(* LS Electric XG5000 project: HS(230517) *)
(* PLC NewPLC *)
(* module base 0 slot 0: FEnet:XGL-EFMT(B) (Fast Ethernet 통신 모듈, 전기 Master) *)
(* module base 1 slot 0: 아날로그입력 모듈:XGF-AC8A (A/D 전류 입력형 8채널) *)
(* module base 1 slot 1: 입력 모듈:XGI-D28A/B (DC 24V 입력, 64점 (전류소스 싱크공용/ 전류소스 입력)) *)
(* module base 1 slot 2: 입력 모듈:XGI-D28A/B (DC 24V 입력, 64점 (전류소스 싱크공용/ 전류소스 입력)) *)
(* module base 1 slot 3: 입력 모듈:XGI-D28A/B (DC 24V 입력, 64점 (전류소스 싱크공용/ 전류소스 입력)) *)
(* module base 1 slot 4: 출력 모듈:XGQ-TR8A/B (트랜지스터 출력, 64점 (0.1A용, 싱크출력/소스출력)) *)
(* module base 1 slot 5: 출력 모듈:XGQ-TR8A/B (트랜지스터 출력, 64점 (0.1A용, 싱크출력/소스출력)) *)
(* module base 1 slot 6: 출력 모듈:XGQ-TR8A/B (트랜지스터 출력, 64점 (0.1A용, 싱크출력/소스출력)) *)
VAR_GLOBAL
    _0100_CH0_ACT AT %UX1.0.16 : BOOL; (* 아날로그입력 모듈: 채널0 운전중 *)
    _0100_CH0_DATA AT %UW1.0.2 : INT; (* 아날로그입력 모듈: 채널0 변환값 *)
    _0100_CH0_IDD AT %UX1.0.160 : BOOL; (* 아날로그입력 모듈: 채널0 입력단선검출 *)
    _0100_CH1_ACT AT %UX1.0.17 : BOOL; (* 아날로그입력 모듈: 채널1 운전중 *)
    _0100_CH1_DATA AT %UW1.0.3 : INT; (* 아날로그입력 모듈: 채널1 변환값 *)
    _0100_CH1_IDD AT %UX1.0.161 : BOOL; (* 아날로그입력 모듈: 채널1 입력단선검출 *)
    _0100_CH2_ACT AT %UX1.0.18 : BOOL; (* 아날로그입력 모듈: 채널2 운전중 *)
    _0100_CH2_DATA AT %UW1.0.4 : INT; (* 아날로그입력 모듈: 채널2 변환값 *)
    _0100_CH2_IDD AT %UX1.0.162 : BOOL; (* 아날로그입력 모듈: 채널2 입력단선검출 *)
    _0100_CH3_ACT AT %UX1.0.19 : BOOL; (* 아날로그입력 모듈: 채널3 운전중 *)
    _0100_CH3_DATA AT %UW1.0.5 : INT; (* 아날로그입력 모듈: 채널3 변환값 *)
    _0100_CH3_IDD AT %UX1.0.163 : BOOL; (* 아날로그입력 모듈: 채널3 입력단선검출 *)
    _0100_CH4_ACT AT %UX1.0.20 : BOOL; (* 아날로그입력 모듈: 채널4 운전중 *)
    _0100_CH4_DATA AT %UW1.0.6 : INT; (* 아날로그입력 모듈: 채널4 변환값 *)
    _0100_CH4_IDD AT %UX1.0.164 : BOOL; (* 아날로그입력 모듈: 채널4 입력단선검출 *)
    _0100_CH5_ACT AT %UX1.0.21 : BOOL; (* 아날로그입력 모듈: 채널5 운전중 *)
    _0100_CH5_DATA AT %UW1.0.7 : INT; (* 아날로그입력 모듈: 채널5 변환값 *)
    _0100_CH5_IDD AT %UX1.0.165 : BOOL; (* 아날로그입력 모듈: 채널5 입력단선검출 *)
    _0100_CH6_ACT AT %UX1.0.22 : BOOL; (* 아날로그입력 모듈: 채널6 운전중 *)
    _0100_CH6_DATA AT %UW1.0.8 : INT; (* 아날로그입력 모듈: 채널6 변환값 *)
    _0100_CH6_IDD AT %UX1.0.166 : BOOL; (* 아날로그입력 모듈: 채널6 입력단선검출 *)
    _0100_CH7_ACT AT %UX1.0.23 : BOOL; (* 아날로그입력 모듈: 채널7 운전중 *)
    _0100_CH7_DATA AT %UW1.0.9 : INT; (* 아날로그입력 모듈: 채널7 변환값 *)
    _0100_CH7_IDD AT %UX1.0.167 : BOOL; (* 아날로그입력 모듈: 채널7 입력단선검출 *)
END_VAR

(* Comments on direct variables
%IX1.1.0	Power On_PB
%IX1.1.1	Power Off_PB
%IX1.1.2	TK1LK_On
%IX1.1.3	출하대 #2_EM
%IX1.1.4	FIRE_EM
SIG
%IX1.1.5	Manual_PB
%IX1.1.6	Auto_PB
%IX1.1.7	TRAIN EM
#1 SIG
%IX1.1.8	TRAIN EM
#2 SIG
%IX1.1.9	TRAIN EM
#3 SIG
%IX1.1.10	TRAIN EM
#4 SIG
%IX1.1.11	BCVF Trouble
%IX1.1.12	AUTO START PB
%IX1.1.13	AUTO Stop PB
%IX1.1.14	LAMP TEST PB
%IX1.1.15	EM-Reset [Panel]
%IX1.1.16	Buffer Tank_EM
%IX1.1.17	Main Tank_EM
%IX1.1.18	출하대 #1_EM
%IX1.1.19	Panel_EM
%IX1.1.20	Scada_선택
%IX1.1.21	Panel_선택
%IX1.1.22	Leakage-1 (L01301) On
%IX1.1.23	VENT1_On
%IX1.1.24	VENT1 Truble_On
%IX1.1.25	TK-001 Clearance
%IX1.1.26	P012A
 OCR & Thermostat
%IX1.1.27	P012A Local key Run[NC]
%IX1.1.28	P012A Stop_PB
%IX1.1.29	P012A Run_PB
%IX1.1.30	P012B
 OCR & Thermostat
%IX1.1.31	P012B Local ready[NC]
%IX1.1.32	P012B Stop_PB
%IX1.1.33	P012B Run_PB
%IX1.1.34	P013
 OCR & Thermostat
%IX1.1.35	P013 Local ready[NC]
%IX1.1.36	P013 Stop_PB
%IX1.1.37	P013 Run_PB
%IX1.1.38	P012A Flow s/w
%IX1.1.39	P012B Flow s/w
%IX1.1.40	P013 Flow Switch
%IX1.1.41	VENT2_On
%IX1.1.42	VENT2 Truble_On
%IX1.1.43	TK-002 Clearance
%IX1.1.44	P021A
 OCR & Thermostat
%IX1.1.45	P021A Local ready[NC]
%IX1.1.46	P021A Stop_PB
%IX1.1.47	P021A Run_PB
%IX1.1.48	P021B
 OCR & Thermostat
%IX1.1.49	P021B Local ready[NC]
%IX1.1.50	P021B Stop_PB
%IX1.1.51	P021B Run_PB
%IX1.1.52	P022
 OCR & Thermostat
%IX1.1.53	P022 Local SW
%IX1.1.54	P022 Stop_PB
%IX1.1.55	P022 Run_PB
%IX1.1.56	P021A Flow Switch
%IX1.1.57	P021B Flow Switch
%IX1.1.58	P022 Flow Switch
%IX1.1.59	TK002_HLV
%IX1.1.60	P012A 1차선택_PB
%IX1.1.61	P012A 2차선택_PB
%IX1.1.62	P012B 1차선택_PB
%IX1.1.63	P012B 2차선택_PB
%IX1.2.0	P021A 1차선택_PB
%IX1.2.1	P021A 2차선택_PB
%IX1.2.2	P021B 1차선택_PB
%IX1.2.3	P021B 2차선택_PB
%IX1.2.4	TK001_HLV
%IX1.2.5	TRANSFER
CLEARANCE
%IX1.2.6	P011A 
OCR & Thermostat
%IX1.2.7	P011A Local ready[NC]
%IX1.2.8	P011A Stop
[Panel]
%IX1.2.9	P011A Run
[Panel]
%IX1.2.10	P011B
 OCR & Thermostat
%IX1.2.11	P011B  Local ready[NC]
%IX1.2.12	P011B Stop_PB
%IX1.2.13	P011B Run_PB
%IX1.2.14	P011C
 OCR & Thermostat
%IX1.2.15	P011C Local ready[NC]
%IX1.2.16	P011C Stop_PB
%IX1.2.17	P011C Run_PB
%IX1.2.18	P011A Flow Switch
%IX1.2.19	P011B Flow Switch
%IX1.2.20	P011C Flow Switch
%IX1.2.21	P011A 1차 선택_PB
%IX1.2.22	P011A 2차선택_PB
%IX1.2.23	P011B 1차 선택_PB
%IX1.2.24	P011B 2차선택_PB
%IX1.2.25	P011C 1차선택_PB
%IX1.2.26	P011C 2차선택_PB
%IX1.2.27	Surge MOV_TR
%IX1.2.28	Surge MOV_LO
%IX1.2.29	Surge Close_PB
%IX1.2.30	Surge 
Close
Position
%IX1.2.31	Surge Open_PB
%IX1.2.32	Surge 
Open Position
%IX1.2.35	RTU-1 Close_PB
%IX1.2.37	RTU-1 Open_PB
%IX1.2.38	RTU-1 MOV_OP
%IX1.2.39	Transfer 수동_운전
%IX1.2.40	Transfer 자동_운전
%IX1.2.41	DR-Tank Water_On
%IX1.2.42	HLVD Close
%IX1.2.43	DRAIN
CLEARANCE
%IX1.2.44	P031
 OCR & Thermostat
%IX1.2.45	P031 Local SW
%IX1.2.46	P031 Stop_PB
%IX1.2.47	P031 Run_PB
%IX1.2.48	R2 PT201A-B 
%IX1.2.49	R3 FT201A-B
%IX1.2.50	R4 PT202A-B
%IX1.2.51	R5 FT202A-B
%IX1.2.52	CAM6_On
%IX1.2.53	드레인 P031_FS
%IX1.2.54	P031 Pressure  SW
%IX1.2.55	LDS ON 
SIG
%IX1.2.56	HLVB(하차 VALVE)
%IX1.2.57	PANTO 1 VPS
%IX1.2.58	PANTO 2 VPS
%IX1.2.59	LDS OFF SIG
%IX1.2.60	LDS EM(HS)
%IX1.2.61	Horn Rest PB
%IX1.3.0	P011A MC On SIG
%IX1.3.1	P011B MC On SIG
%IX1.3.2	P011C MC On SIG
%IX1.3.3	P012A MC On SIG
%IX1.3.4	P012B MC On SIG
%IX1.3.5	P013 MC On SIG
%IX1.3.6	P021A MC ON SIG
%IX1.3.7	P021B MC On SIG
%IX1.3.8	P022 MC On SIG
%IX1.3.9	DRAIN MC On SIG
%ID1.0.0	디지털_입력
%QX1.4.0	Power On_Lamp
%QX1.4.1	Power Off_Lamp
%QX1.4.2	Panel 선택 Lamp
%QX1.4.3	Scada 선택 Lamp
%QX1.4.4	TK3 누유 Lamp
%QX1.4.5	Manual_Lamp
%QX1.4.6	Auto_Lamp
%QX1.4.7	Auto Start Lamp
%QX1.4.8	Auto Stop Lamp
%QX1.4.9	Leakage TK-001 Lamp
%QX1.4.10	Leakage TK-002 Lamp
%QX1.4.11	Leakage TK-003 Lamp
%QX1.4.12	EM TK01 (BUFFER) Lamp
%QX1.4.13	EM TK02 (MAIN) Lamp
%QX1.4.14	Lamp Test Lamp
%QX1.4.15	PANTO 1  EM LAMP
%QX1.4.16	Horn Stop Lamp
%QX1.4.17	EM Panel Lamp
%QX1.4.18	PANTO 2 EM LAMP
%QX1.4.19	FIRE_EM
LAMP
%QX1.4.22	PIT201A Trouble Lamp
%QX1.4.23	PIT201B Trouble Lamp
%QX1.4.24	CVP OPEN LAMP
%QX1.4.25	EV OPEN LAMP
%QX1.4.26	PIT202A Trouble Lamp
%QX1.4.27	PIT202B Trouble Lamp
%QX1.4.28	FIT3 Trouble Lamp
%QX1.4.29	FIT4 Trouble Lamp
%QX1.4.30	Master_Plc Lamp
%QX1.4.31	Standby_  Plc Lamp
%QX1.4.32	EM-Stop Reset Lamp
%QX1.4.33	Leakage-1 Lamp
%QX1.4.34	VENT1 Trouble Lamp
%QX1.4.35	VENT1 Run Lamp
%QX1.4.36	P012A Trouble Lamp
%QX1.4.37	P012A Local Lamp
%QX1.4.38	P012A Stop Lamp
%QX1.4.39	P012A Run Lamp
%QX1.4.40	P012B Trouble Lamp
%QX1.4.41	P012B Local Lamp
%QX1.4.42	P012B Stop Lamp
%QX1.4.43	P012B Run Lamp
%QX1.4.44	P013 Trouble Lamp
%QX1.4.45	P013 Local Lamp
%QX1.4.46	P013 Stop Lamp
%QX1.4.47	P013 Run Lamp
%QX1.4.48	TK-001 Level_HH
%QX1.4.49	TK-001 Level_H
%QX1.4.50	TK-001 ATG TROUBLE
%QX1.4.51	TK-001 Level_L
%QX1.4.52	TK-001 Level_LL
%QX1.4.53	VENT2 Trouble Lamp
%QX1.4.54	VENT2 Run Lamp
%QX1.4.55	P021A Trouble Lamp
%QX1.4.56	P021A Local Lamp
%QX1.4.57	P021A Stop Lamp
%QX1.4.58	P021A Run Lamp
%QX1.4.59	P021B Trouble Lamp
%QX1.4.60	P021B Local Lamp
%QX1.4.61	P021B Stop Lamp
%QX1.4.62	P021B Run Lamp
%QX1.4.63	P022 Trouble Lamp
%QX1.5.0	P022 Local Lamp
%QX1.5.1	P022 Stop Lamp
%QX1.5.2	P022 Run Lamp
%QX1.5.3	TK-002 Level_HH
%QX1.5.4	TK-002 Level_H
%QX1.5.5	TK-002 ATG TROUBLE
%QX1.5.6	TK-002 Level_L
%QX1.5.7	TK-002 Level_LL
%QX1.5.8	HLV 01301 Lamp
%QX1.5.9	P012A 1차 선택 Lamp
%QX1.5.10	P012A 2차 선택 Lamp
%QX1.5.11	P012B 1차 선택 Lamp
%QX1.5.12	P012B 2차 선택 Lamp
%QX1.5.13	P021A 1차 선택 Lamp
%QX1.5.14	P021A 2차 선택 Lamp
%QX1.5.15	P021B 1차 선택 Lamp
%QX1.5.16	P021B 2차 선택 Lamp
%QX1.5.17	TK-001 HLV_Out
%QX1.5.18	P011A Trouble Lamp
%QX1.5.19	P011A Local Lamp
%QX1.5.20	P011A Stop Lamp
%QX1.5.21	P011A Run Lamp
%QX1.5.22	P011B Trouble Lamp
%QX1.5.23	P011B Local Lamp
%QX1.5.24	P011B Stop Lamp
%QX1.5.25	P011B Run Lamp
%QX1.5.26	P011C Trouble Lamp
%QX1.5.27	P011C Local Lamp
%QX1.5.28	P011C Stop Lamp
%QX1.5.29	P011C Run Lamp
%QX1.5.30	P011A 1차 선택 Lamp
%QX1.5.31	P011A 2차 선택 Lamp
%QX1.5.32	P011B 1차 선택 Lamp
%QX1.5.33	P011B 2차 선택 Lamp
%QX1.5.34	P011C 1차 선택 Lamp
%QX1.5.35	P011C 2차 선택 Lamp
%QX1.5.36	Surge Trouble Lamp
%QX1.5.38	Surge Close Lamp
%QX1.5.39	Surge 
Open Lamp
%QX1.5.40	RTU-1 Trouble Lamp
%QX1.5.41	RTU-1 Local Lamp
%QX1.5.42	RTU-1 Close Lamp
%QX1.5.43	RTU-1 Open Lamp
%QX1.5.44	Transfer 수동 LAMP
%QX1.5.45	Transfer 자동 LAMP
%QX1.5.46	600GPM LAMP
%QX1.5.47	1200GPM LAMP
%QX1.5.48	POLPRV LAMP
%QX1.5.49	RTU#1 OPEN LAMP
%QX1.5.50	RTU#2 OPEN LAMP
%QX1.5.51	RTU#3 OPEN LAMP
%QX1.5.52	RTU#4 OPEN LAMP
%QX1.5.53	RTU#5 OPEN LAMP
%QX1.5.54	Drain Water Lamp
%QX1.5.55	Drain HLVD_Full Lamp
%QX1.5.56	P031 Trouble Lamp
%QX1.5.57	P031 Local Lamp
%QX1.5.58	P031 Stop Lamp
%QX1.5.59	P031 Run Lamp
%QX1.5.60	TK-003 Level_HH
%QX1.5.61	TK-003 Level_H
%QX1.5.62	TK-003 ATG TROUBLE
%QX1.5.63	TK-003 Level_L
%QX1.6.0	TK-003 Level_LL
%QX1.6.1	CVP_Sol
%QX1.6.2	EV_Sol
%QX1.6.3	P011A_CVTF
%QX1.6.4	P011B_CVTF
%QX1.6.5	P011C_CVTF
%QX1.6.6	P-011A MCC_Run
%QX1.6.7	P-011B MCC_Run
%QX1.6.8	P-011C MCC_Run
%QX1.6.9	P-012A MCC_Run
%QX1.6.10	P-012B MCC_Run
%QX1.6.11	P-013 MCC_Run
%QX1.6.12	TK-001 HLV_Sol
%QX1.6.13	P-021A MCC_Run
%QX1.6.14	P-021B MCC_Run
%QX1.6.15	P-022 MCC_Run
%QX1.6.16	TK-001 HLV_Sol
%QX1.6.17	P-031 MCC_Run
%QX1.6.18	TK-003 HLVD_Out
%QX1.6.19	Surge Valve Open
%QX1.6.20	Surge Valve Close 
%QX1.6.21	RMOR
%QX1.6.22	RMCR
%QX1.6.23	Horn_Relay
%QX1.6.24	CVPl Lamp
%QX1.6.25	EV Lamp
%QX1.6.26	SURGE MOV
CLOSE SIG
%QX1.6.27	TRANSFER PUMP RUN
SIG
%QX1.6.28	SURGE MOV
OPEN SIG
%QX1.6.34	TO LDS
[SURGE CLOSE]
%QX1.6.35	TO LDS
[SURGE OPEN]
%QX1.6.36	TO LDS
[TP ALARM]
%QX1.6.37	LDS PUMP STOP SIG
%MX0	출하압력 Min
%MX1	TK01_EM
%MX2	TK02_EM
%MX3	PANTO 1 EM
%MX4	Panel_EM
%MX5	Total Em 
%MX6	Total Alarm
%MX7	Horn_Stop
%MX8	Horn Stop   Lamp   (SCADA)
%MX9	EM-Stop Reset   Lamp   (SCADA)
%MX10	P011A Pump Stop Set
%MX11	P011B Pump Stop Set
%MX12	P011C Pump Stop Set
%MX13	P012A Pump Stop Set
%MX14	P012B Pump Stop Set
%MX15	P013 Pump Stop Set
%MX16	LDS_EM(HS)
%MX17	LDS_EM
(POL)
%MX18	NMR5000_ERR
%MX19	FIRE_EM
%MX20	POL 수령탱크 HH
%MX21	P021A Pump Stop Set
%MX22	P021B Pump Stop Set
%MX23	P022 Pump Stop Set
%MX24	P031 Pump Stop Set
%MX25	P011A Lock key Run
%MX26	P011B Lock key Run
%MX27	P011C Lock key Run
%MX28	P012A Lock key Run
%MX29	P012B Lock key Run
%MX30	P013 Lock key Run
%MX31	P021A Lock key Run
%MX32	P021B Lock key Run
%MX33	P022 Lock key Run
%MX34	P031 Lock key Run
%MX41	POL TO RTU#1 ON SIG
%MX42	POL TO RTU#2 ON SIG
%MX43	POL TO RTU#3 ON SIG
%MX44	POL TO RTU#4 ON SIG
%MX45	POL TO RTU#5 ON SIG
%MX64	from SCADA  Manual [Select]
%MX65	from SCADA Auto [Select]
%MX66	AUTO START (SCADA)
%MX67	AUTO Stop PB(Scada)
%MX68	EM-Reset [SCADA]
%MX69	Horn Reset SCADA
%MX76	F03 Auto On_Out
%MX77	F03 Manual On_PB
%MX78	F03 Manual On_Out
%MX79	F01 Alam_Reset
%MX80	TRAIN EM
#1
%MX81	TRAIN EM
#2
%MX82	TRAIN EM
#3
%MX83	TRAIN EM
#4
%MX100	CH0 단선검출
%MX101	CH1 단선검출
%MX102	CH2 단선검출
%MX103	CH3 단선검출
%MX104	CH4 단선검출
%MX105	CH5 단선검출
%MX106	CH6 단선검출
%MX107	CH7 단선검출
%MX128	P011A Run [SCADA]
%MX129	P011A Stop
[SCADA]
%MX132	P011B Run [SCADA]
%MX133	P011B Stop_PB Scada
%MX136	P011C Run_PB Scada
%MX137	P011B Stop_PB Scada
%MX140	P012A Run_PB Scada
%MX141	P012A Stop_PB Scada
%MX144	P012B Run_PB Scada
%MX145	P012B Stop_PB Scada
%MX148	P013 Run_PB Scada
%MX149	P013 Stop_PB Scada
%MX152	P021A Run_PB Scada
%MX153	P021A Stop_PB Scada
%MX156	P021B Run_PB Scada
%MX157	P021B Stop_PB Scada
%MX160	P022 Run_PB Scada
%MX161	P022 Stop_PB Scada
%MX164	P031 Run_PB Scada
%MX165	P031 Stop_PB Scada
%MX266	MOV M01201 OPEN
%MX267	MOV M01201 CLOSE
%MX310	TK-001 Level_HH
%MX311	TK-001 Level_H
%MX312	TK-001 ATG TROUBLE SIG
%MX313	TK-001 Level_L
%MX314	TK-001 Level_LL
%MX320	TK-002 Level_HH
%MX321	TK-002 Level_H
%MX322	TK-002 ATG TROUBLE SIG
%MX323	TK-002 Level_L
%MX324	TK-002 Level_LL
%MX325	POL TOTAL EM (POL ->SCADA ->HS)
%MX330	TK-003 Level_HH
%MX331	TK-003 Level_H
%MX332	TK-003 ATG TROUBLE SIG
%MX333	TK-003 Level_L
%MX334	TK-003 Level_LL
%MX340	P011A 선택 SET
%MX341	P011B 선택 SET
%MX342	P011C 선택 SET
%MX343	P011A 2차 선택
%MX344	P011B 2차 선택
%MX345	P011C 2차 선택
%MX346	P011A 선택 SIG
%MX347	P011B 선택 SIG
%MX348	P011C 선택 SIG
%MX350	P012A 1차 선택
%MX351	P012B 1차 선택
%MX352	P012A 2차 선택
%MX353	P012B 2차 선택
%MX360	P021A 1차 선택
%MX361	P021B 1차 선택
%MX362	P021A 2차 선택
%MX363	P021B 2차 선택
%MX364	RTU1 OPEN LAMP (LDS->PLC)
%MX365	RTU2 OPEN LAMP (LDS->PLC)
%MX366	RTU3 OPEN LAMP (LDS->PLC)
%MX367	RTU4 OPEN LAMP (LDS->PLC)
%MX368	RTU5 OPEN LAMP (LDS->PLC)
%MX402	TK-110 ATG Trouble
%MX448	P011A  1차 선택 SWITCH  (SCADA)
%MX449	P011B 1차 선택 SWITCH  (SCADA)
%MX450	P011C 1차 선택 SWITCH  (SCADA)
%MX451	P011A  2차 선택 SWITCH  (SCADA)
%MX452	P011B 2차 선택 SWITCH  (SCADA)
%MX453	P011C 2차 선택 SWITCH  (SCADA)
%MX457	선택완료  (SCADA)
%MX458	P012A  1차 선택 SWITCH  (SCADA)
%MX459	P012B  1차 선택 SWITCH  (SCADA)
%MX460	P012A  2차 선택 SWITCH  (SCADA)
%MX461	P012B  2차 선택 SWITCH  (SCADA)
%MX467	선택완료  (SCADA)
%MX468	P021A  1차 선택 SWITCH  (SCADA)
%MX469	P021B 1차 선택 SWITCH  (SCADA)
%MX470	P021A  2차 선택 SWITCH  (SCADA)
%MX471	P021B 2차 선택 SWITCH  (SCADA)
%MX472	선택 완료    (SCADA)
%MX473	LDS 누유
%MX474	LDS  EM(POL)
%MX475	이송펌프 선택 초기화
%MX477	선택완료  (SCADA)
%MX960	P011A FS SIG
%MX961	P011B FS SIG
%MX962	P011C FS SIG
%MX963	P012A FS SIG
%MX964	P012B FS SIG
%MX965	P013 FS SIG
%MX966	P021A FS SIG
%MX967	P021B FS SIG
%MX968	P022 FS SIG
%MX969	P031 FS SIG
%MX1000	TK-002 MAIN TANK 누유
%MX1001	TK-001 BUFFER TANK 누유
%MX1002	TK-003 DRAIN TANK 누유
%MX6400	Panel Manual [Select]
%MX6401	SCADA  Manual [Select]
%MX6402	Panel   Auto [Select]
%MX6403	SCADA  Auto [Select]
%MX6410	Manual Select
[to SCADA]
%MX6411	Auto Select
[to SCADA]
%MX6464	LAMP TEST SIG
%MX6478	임시
%MX12800	PANTO 2 EM
%MX19200	P011A  Alarm
%MX19201	P011B  Alarm
%MX19202	P011C  Alarm
%MX19203	P012A  Alarm
%MX19204	P012B  Alarm
%MX19205	P013  Alarm
%MX19206	P021A  Alarm
%MX19207	P021B  Alarm
%MX19208	P022  Alarm
%MX19209	P031 Alarm
%MX19210	Surge Mov M01201 Trouble
%MX19211	RTU-1 Trouble Lamp(SCADA)
%MX19212	PIT201A Trouble   Lamp   (SCADA)
%MX19213	PIT201B Trouble   Lamp   (SCADA)
%MX19214	FIT201A Trouble   Lamp   (SCADA)
%MX19215	FIT201B Trouble   Lamp  (SCADA)
%MX19216	PIT202A Trouble   Lamp   (SCADA)
%MX19217	PIT202B Trouble   Lamp   (SCADA)
%MX19218	FIT3 Trouble   Lamp  (SCADA)
%MX19219	FIT4 Trouble   Lamp  (SCADA)
%MX19264	P011A RUN SIG
%MX19265	P011B 수동 RUN
%MX19266	P011C 수동 RUN
%MX19267	P012A 수동 RUN
%MX19268	P012B 수동 RUN
%MX19269	P013 수동 RUN
%MX19270	P021A 수동 RUN
%MX19271	P021B 수동 RUN
%MX19272	P022 수동 RUN
%MX19273	P031 수동 RUN
%MX19274	MOV 01201 OPEN 
%MX19275	MOV 01201 CLOSE
%MX19328	P011A FS ALARM
%MX19329	P011B FS ALARM
%MX19330	P011C FS ALARM
%MX19331	P012A FS ALARM
%MX19332	P012B FS ALARM
%MX19333	P013 FS ALARM
%MX19334	P021A FS ALARM
%MX19335	P021B FS ALARM
%MX19336	P022 FS ALARM
%MX19337	P031 FS ALARM
%MX23680	MAIN TANK 수령 송유관 색변화
%MX23681	MAIN TANK  불출 송유관 색변화
%MX23682	MAIN TANK  드레인 송유관 색변화 
%MX23683	BUFFER TANK  이송(BPCV) 송유관 색변화
%MX23684	BUFFER TANK이송  (CVTF1) 송유관 색변화
%MX23685	BUFFER TANK이송  (CVTF2) 송유관 색변화 2
%MX23686	BUFFER TANK이송  (CVTF3) 송유관 색변화
%MX23687	BUFFER TANK이송  (P012A,B) 송유관 색변화
%MX23688	BUFFER TANK회수 송유관 색변화1 
%MX23689	BUFFER TANK회수 송유관 색변화 2
%MX23691	BUFFER TANK DRAIN 송유관 색변화
%MX23692	BUFFER TANK 하차 송유관 색변화
%MX23693	DRAIN TANK DRAIN 송유관 색변화 5
%MX23694	PANTO1 송유관 색변화
%MX23695	PANTO02 송유관 색변화
%MX23696	이송 MAIN 송유관 색변화 
%MX23697	BUFFER & MAIN TANK DRAIN 송유관 색변화
%MX25600	AUTO START OK
%MX25601	AUTO START SIG
%MX25602	ALL REMOTE
%MX25603	AUTO START
%WB20	FROM POL
[HIGH 8 BIT]
%WB21	FROM POL
[LOW 8 BIT]
%WW0	TK-001 HH SET
%WW1	TK-001 H SET
%WW2	TK-001 L SET
%WW3	TK-001 LL SET
%WW4	TK-002 HH SET
%WW5	TK-002 H SET
%WW6	TK-002 L SET
%WW7	TK-002 LL SET
%WW9	FROM POL [16 BIT]
%WW10	이송 PUMP P011 1차 선택 SET
%WW11	이송 PUMP P011 2차 선택 SET
%WW12	이송 PUMP P012 1차 선택 SET
%WW13	이송 PUMP P012B  2차선택 SET
%WW14	이송 PUMP P021A  운전 선택 SET
%WW15	이송 PUMP P021B  운전 선택 SET
%WW20	TANK101 문자열
%WW21	TANK102 문자열
%WW22	TANK103 문자열
%WW30	TK-003 HH SET
%WW31	TK-003 H SET
%WW32	TK-003 L SET
%WW33	TK-003 LL SET
%WW34	P011 펌프 선택
%WW100	PT01 변환값
%WW102	PT01  이송압력 PSI
%WW150	P011A RUN SET
%WW151	P011B RUN SET
%WW152	P011C RUN SET
%WW153	P012A RUN SET
%WW154	P012B RUN SET
%WW155	P013 RUN SET
%WW156	P021A RUN SET
%WW157	P021B RUN SET
%WW158	P022 RUN SET
%WW159	P031 RUN SET
%WW160	MOV 01201 OPEN SET
%WW200	FT01 변환값
%WW202	FT01  이송유량 GPM
%WW300	PT02 변환값
%WW302	PT02  송유압력 PSI
%WW400	FT02 변환값
%WW402	FT02  이송유량 GPM
%WW500	DRAIN TANK 변환값
%WW506	DRAIN TANK LEVEL (PLC -> SCADA)
%WW600	MAIN TANK 변환값
%WW700	BUFFER TANK 변환값
%WW709	TK-110 ATG TROUBLE
%WW800	DRAIN TANK 변환값
%WW1000	TK-001 LEVEL 
(NMR TO PLC)
%WW1001	TK-001 ATG Trouble
%WW1003	TK-002 LEVEL (PLC->SCADA)
%WW1004	TK-002 ATG Trouble
*)

PROGRAM Main (* task: 스캔 프로그램 *)
VAR
    L_TST : TON;
    L_TST_FS : TON;
END_VAR

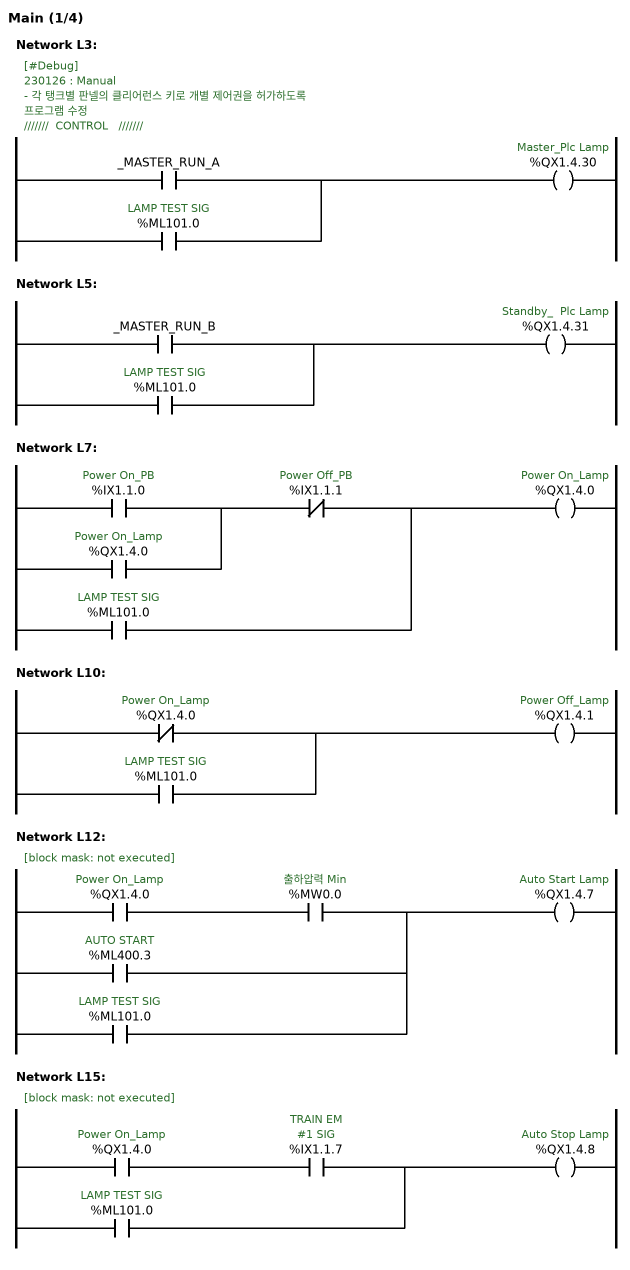
(* [#Debug] *)
(* 230126 : Manual / - 각 탱크별 판넬의 클리어런스 키로 개별 제어권을 허가하도록 / 프로그램 수정 *)
(* ///////  CONTROL   /////// *)
(* Rung L3 *)
%QX1.4.30 := _MASTER_RUN_A OR %ML101.0;
(* Rung L5 *)
%QX1.4.31 := _MASTER_RUN_B OR %ML101.0;
(* Rung L7 *)
%QX1.4.0 := ((%IX1.1.0 OR %QX1.4.0) AND NOT %IX1.1.1) OR %ML101.0;
(* Rung L10 *)
%QX1.4.1 := NOT %QX1.4.0 OR %ML101.0;
(* Rung L12 is block-masked: not executed *)
// %QX1.4.7 := (%QX1.4.0 AND %MW0.0) OR %ML400.3 OR %ML101.0;
(* Rung L15 is block-masked: not executed *)
// %QX1.4.8 := (%QX1.4.0 AND %IX1.1.7) OR %ML101.0;

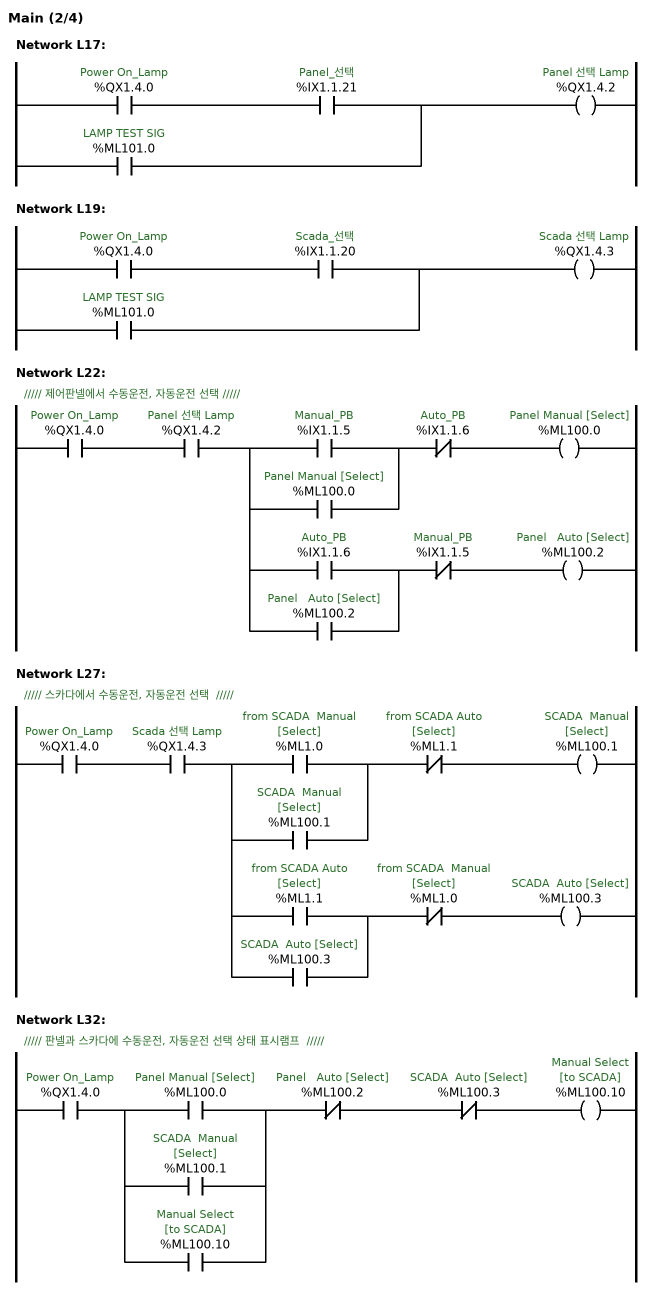
(* Rung L17 *)
%QX1.4.2 := (%QX1.4.0 AND %IX1.1.21) OR %ML101.0;
(* Rung L19 *)
%QX1.4.3 := (%QX1.4.0 AND %IX1.1.20) OR %ML101.0;
(* ///// 제어판넬에서 수동운전, 자동운전 선택 ///// *)
(* Rung L22 *)
%ML100.0 := %QX1.4.0 AND %QX1.4.2 AND (%IX1.1.5 OR %ML100.0) AND NOT %IX1.1.6;
%ML100.2 := %QX1.4.0 AND %QX1.4.2 AND (%IX1.1.6 OR %ML100.2) AND NOT %IX1.1.5;
(* ///// 스카다에서 수동운전, 자동운전 선택  ///// *)
(* Rung L27 *)
%ML100.1 := %QX1.4.0 AND %QX1.4.3 AND (%ML1.0 OR %ML100.1) AND NOT %ML1.1;
%ML100.3 := %QX1.4.0 AND %QX1.4.3 AND (%ML1.1 OR %ML100.3) AND NOT %ML1.0;
(* ///// 판넬과 스카다에 수동운전, 자동운전 선택 상태 표시램프  ///// *)
(* Rung L32 *)
%ML100.10 := %QX1.4.0 AND (%ML100.0 OR %ML100.1 OR %ML100.10) AND NOT %ML100.2 AND NOT %ML100.3;

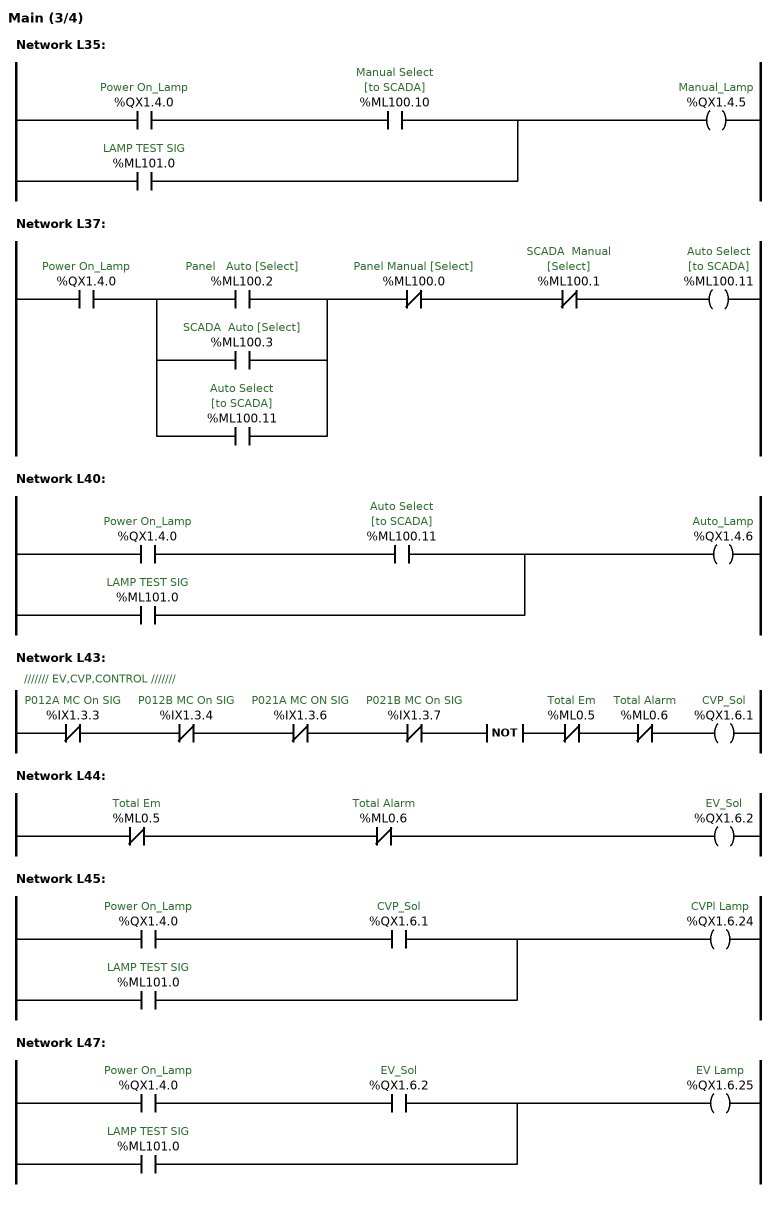
(* Rung L35 *)
%QX1.4.5 := (%QX1.4.0 AND %ML100.10) OR %ML101.0;
(* Rung L37 *)
%ML100.11 := %QX1.4.0 AND (%ML100.2 OR %ML100.3 OR %ML100.11) AND NOT %ML100.0 AND NOT %ML100.1;
(* Rung L40 *)
%QX1.4.6 := (%QX1.4.0 AND %ML100.11) OR %ML101.0;
(* /////// EV,CVP,CONTROL /////// *)
(* Rung L43 *)
%QX1.6.1 := NOT (NOT %IX1.3.3 AND NOT %IX1.3.4 AND NOT %IX1.3.6 AND NOT %IX1.3.7) AND NOT %ML0.5 AND NOT %ML0.6;
(* Rung L44 *)
%QX1.6.2 := NOT %ML0.5 AND NOT %ML0.6;
(* Rung L45 *)
%QX1.6.24 := (%QX1.4.0 AND %QX1.6.1) OR %ML101.0;
(* Rung L47 *)
%QX1.6.25 := (%QX1.4.0 AND %QX1.6.2) OR %ML101.0;

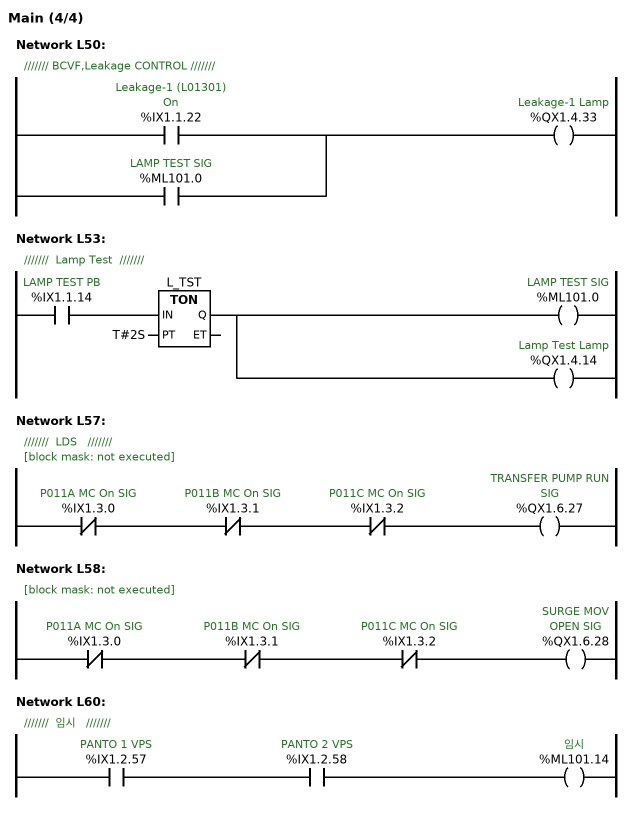
(* /////// BCVF,Leakage CONTROL /////// *)
(* Rung L50 *)
%QX1.4.33 := %IX1.1.22 OR %ML101.0;
(* ///////  Lamp Test  /////// *)
(* Rung L53 *)
L_TST(IN := %IX1.1.14, PT := T#2S);
%ML101.0 := L_TST.Q;
%QX1.4.14 := L_TST.Q;
(* ///////  LDS   /////// *)
(* Rung L57 is block-masked: not executed *)
// %QX1.6.27 := NOT %IX1.3.0 AND NOT %IX1.3.1 AND NOT %IX1.3.2;
(* Rung L58 is block-masked: not executed *)
// %QX1.6.28 := NOT %IX1.3.0 AND NOT %IX1.3.1 AND NOT %IX1.3.2;
(* ///////  임시   /////// *)
(* Rung L60 *)
%ML101.14 := %IX1.2.57 AND %IX1.2.58;
END_PROGRAM

PROGRAM Manual (* task: 스캔 프로그램 *)
VAR
    INST : TP; (* PUMP FS 떨림방지 *)
    INST1 : TP; (* PUMP FS 떨림방지 *)
    P011A_FS : TON;
    P011B_FS : TON;
    P011C_FS : TON;
    P012A_FS : TON;
    P012B_FS : TON;
    P012C_FS : TON;
    P013B_FS : TON;
    P013C_FS : TON;
    P013_FS : TON;
    P014_FS : TON;
    P021A_FS : TON;
    P022A_FS : TON;
    P022_FS : TON;
    P023_FS : TON;
    P031_FS : TON;
    P031_run : TON;
    P031_압력SW : TON;
    P032_FS : TON;
    P033_FS : TON;
    P034_FS : TON;
    P1O1B_FS : TON;
    P1O2B_FS : TON;
    P1O3B_FS : TON;
    TK031_HLV_Pressure_Charging : TON; (* 드레인탱크 031 HLVD 작동을 위한 상시 가압 탱크에 압력을 자체 충전하기위한 압력 감지 접점이 작동하면 펌프를 0.5초 지연 후 작동시킨다 *)
END_VAR
VAR_EXTERNAL
    _0100_CH2_DATA : INT; (* AT %UW1.0.4 *) (* 아날로그입력 모듈: 채널2 변환값 *)
    _0100_CH3_DATA : INT; (* AT %UW1.0.5 *) (* 아날로그입력 모듈: 채널3 변환값 *)
    _0100_CH4_ACT : BOOL; (* AT %UX1.0.20 *) (* 아날로그입력 모듈: 채널4 운전중 *)
    _0100_CH4_DATA : INT; (* AT %UW1.0.6 *) (* 아날로그입력 모듈: 채널4 변환값 *)
    _0100_CH5_ACT : BOOL; (* AT %UX1.0.21 *) (* 아날로그입력 모듈: 채널5 운전중 *)
    _0100_CH5_DATA : INT; (* AT %UW1.0.7 *) (* 아날로그입력 모듈: 채널5 변환값 *)
    _0100_CH6_ACT : BOOL; (* AT %UX1.0.22 *) (* 아날로그입력 모듈: 채널6 운전중 *)
    _0100_CH6_DATA : INT; (* AT %UW1.0.8 *) (* 아날로그입력 모듈: 채널6 변환값 *)
    _0100_CH7_ACT : BOOL; (* AT %UX1.0.23 *) (* 아날로그입력 모듈: 채널7 운전중 *)
    _0100_CH7_DATA : INT; (* AT %UW1.0.9 *) (* 아날로그입력 모듈: 채널7 변환값 *)
END_VAR
VAR
    _e1 : R_TRIG;
    _e2 : R_TRIG;
END_VAR

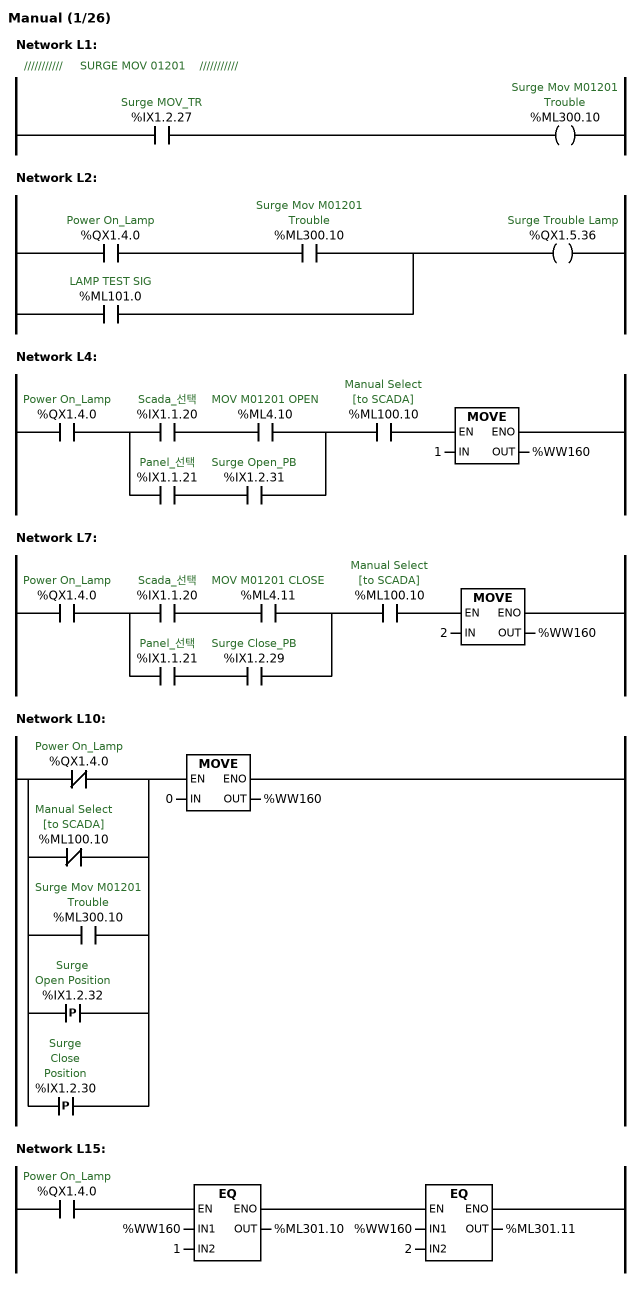
(* ///////////     SURGE MOV 01201    /////////// *)
(* Rung L1 *)
%ML300.10 := %IX1.2.27;
(* Rung L2 *)
%QX1.5.36 := (%QX1.4.0 AND %ML300.10) OR %ML101.0;
(* Rung L4 *)
IF %QX1.4.0 AND ((%IX1.1.20 AND %ML4.10) OR (%IX1.1.21 AND %IX1.2.31)) AND %ML100.10 THEN
    %WW160 := 1;
END_IF;
(* Rung L7 *)
IF %QX1.4.0 AND ((%IX1.1.20 AND %ML4.11) OR (%IX1.1.21 AND %IX1.2.29)) AND %ML100.10 THEN
    %WW160 := 2;
END_IF;
(* Rung L10 *)
_e1(CLK := %IX1.2.32);
_e2(CLK := %IX1.2.30);
IF NOT %QX1.4.0 OR NOT %ML100.10 OR %ML300.10 OR _e1.Q OR _e2.Q THEN %WW160 := 0; END_IF;
(* Rung L15 *)
IF %QX1.4.0 THEN
    %ML301.10 := %WW160 = 1;
    %ML301.11 := %WW160 = 2;
END_IF;

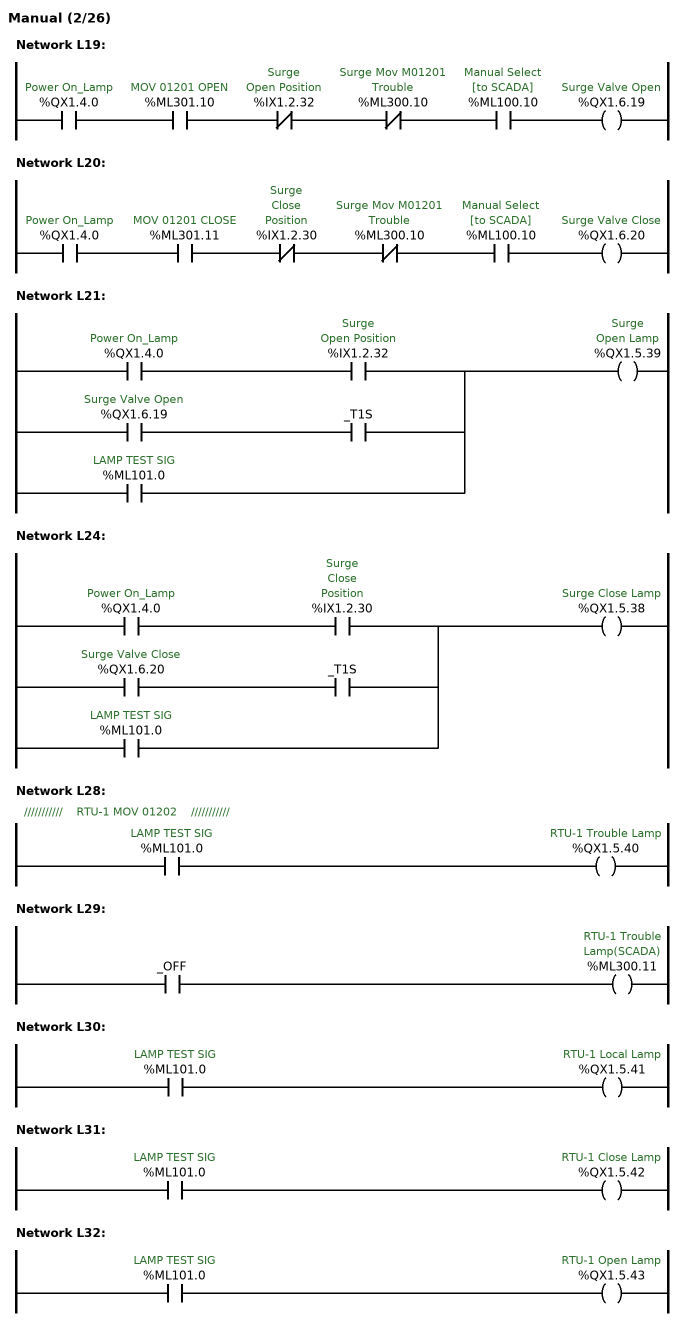
(* Rung L19 *)
%QX1.6.19 := %QX1.4.0 AND %ML301.10 AND NOT %IX1.2.32 AND NOT %ML300.10 AND %ML100.10;
(* Rung L20 *)
%QX1.6.20 := %QX1.4.0 AND %ML301.11 AND NOT %IX1.2.30 AND NOT %ML300.10 AND %ML100.10;
(* Rung L21 *)
%QX1.5.39 := (%QX1.4.0 AND %IX1.2.32) OR (%QX1.6.19 AND _T1S) OR %ML101.0;
(* Rung L24 *)
%QX1.5.38 := (%QX1.4.0 AND %IX1.2.30) OR (%QX1.6.20 AND _T1S) OR %ML101.0;
(* ///////////    RTU-1 MOV 01202    /////////// *)
(* Rung L28 *)
%QX1.5.40 := %ML101.0;
(* Rung L29 *)
%ML300.11 := _OFF;
(* Rung L30 *)
%QX1.5.41 := %ML101.0;
(* Rung L31 *)
%QX1.5.42 := %ML101.0;
(* Rung L32 *)
%QX1.5.43 := %ML101.0;

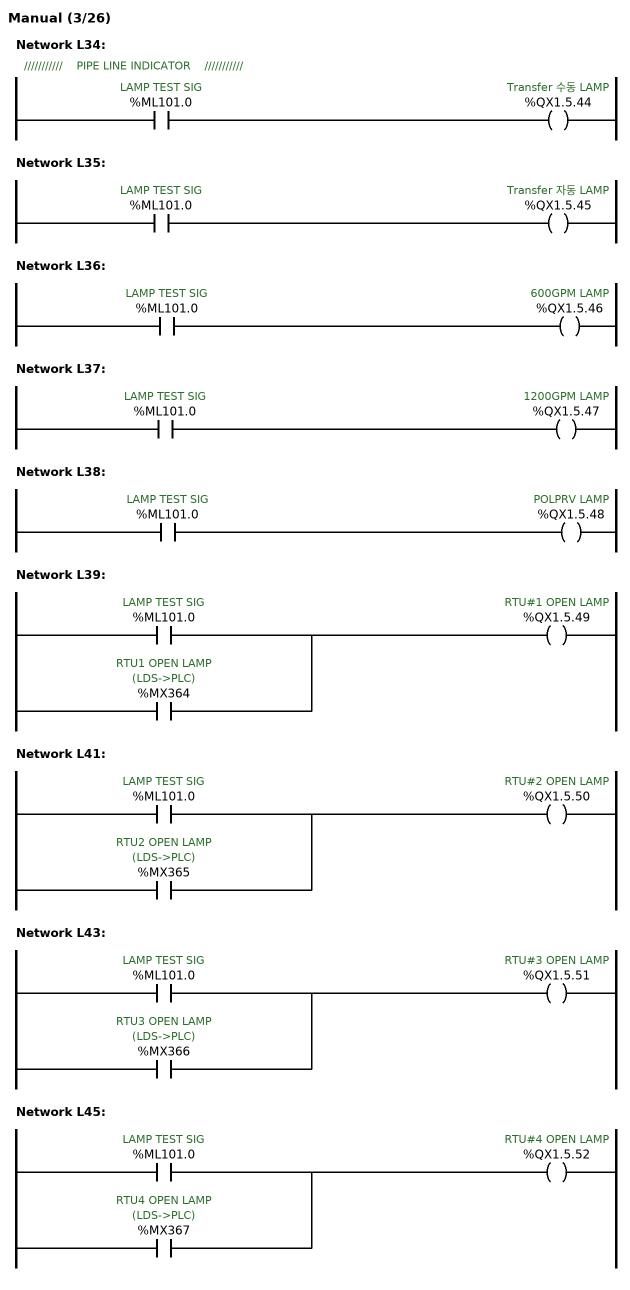
(* ///////////    PIPE LINE INDICATOR    /////////// *)
(* Rung L34 *)
%QX1.5.44 := %ML101.0;
(* Rung L35 *)
%QX1.5.45 := %ML101.0;
(* Rung L36 *)
%QX1.5.46 := %ML101.0;
(* Rung L37 *)
%QX1.5.47 := %ML101.0;
(* Rung L38 *)
%QX1.5.48 := %ML101.0;
(* Rung L39 *)
%QX1.5.49 := %ML101.0 OR %MX364;
(* Rung L41 *)
%QX1.5.50 := %ML101.0 OR %MX365;
(* Rung L43 *)
%QX1.5.51 := %ML101.0 OR %MX366;
(* Rung L45 *)
%QX1.5.52 := %ML101.0 OR %MX367;

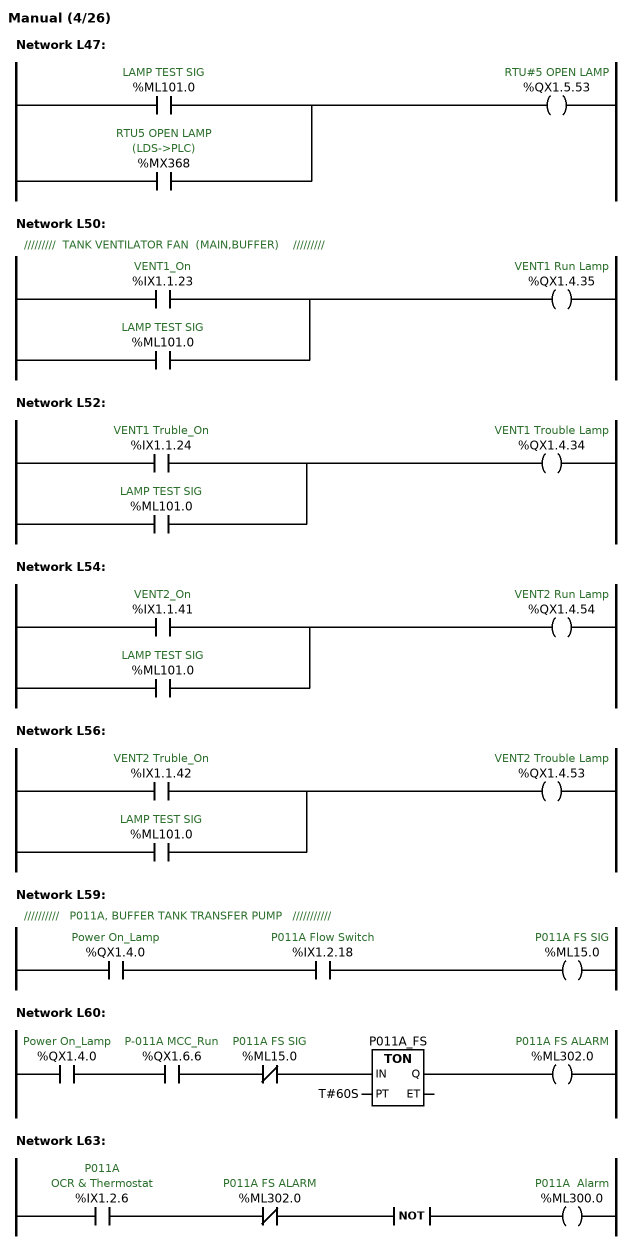
(* Rung L47 *)
%QX1.5.53 := %ML101.0 OR %MX368;
(* /////////  TANK VENTILATOR FAN  (MAIN,BUFFER)    ///////// *)
(* Rung L50 *)
%QX1.4.35 := %IX1.1.23 OR %ML101.0;
(* Rung L52 *)
%QX1.4.34 := %IX1.1.24 OR %ML101.0;
(* Rung L54 *)
%QX1.4.54 := %IX1.1.41 OR %ML101.0;
(* Rung L56 *)
%QX1.4.53 := %IX1.1.42 OR %ML101.0;
(* //////////   P011A, BUFFER TANK TRANSFER PUMP   /////////// *)
(* Rung L59 *)
%ML15.0 := %QX1.4.0 AND %IX1.2.18;
(* Rung L60 *)
P011A_FS(IN := %QX1.4.0 AND %QX1.6.6 AND NOT %ML15.0, PT := T#60S);
%ML302.0 := P011A_FS.Q;
(* Rung L63 *)
%ML300.0 := NOT (%IX1.2.6 AND NOT %ML302.0);

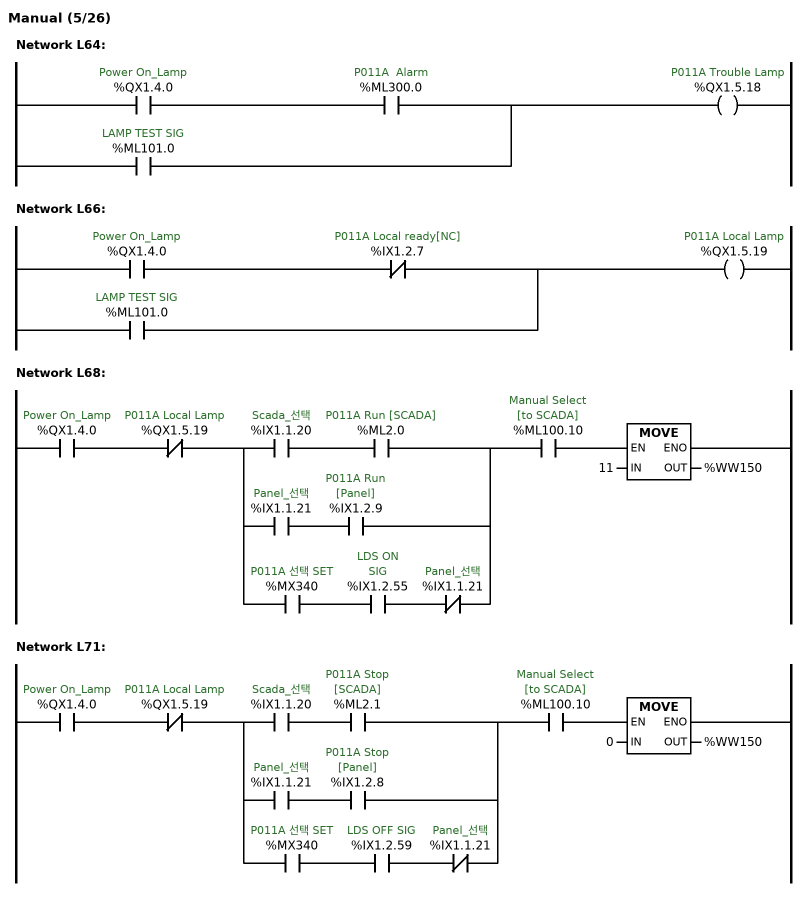
(* Rung L64 *)
%QX1.5.18 := (%QX1.4.0 AND %ML300.0) OR %ML101.0;
(* Rung L66 *)
%QX1.5.19 := (%QX1.4.0 AND NOT %IX1.2.7) OR %ML101.0;
(* Rung L68 *)
IF %QX1.4.0 AND NOT %QX1.5.19 AND ((%IX1.1.20 AND %ML2.0) OR (%IX1.1.21 AND %IX1.2.9) OR (%MX340 AND %IX1.2.55 AND NOT %IX1.1.21)) AND %ML100.10 THEN
    %WW150 := 11;
END_IF;
(* Rung L71 *)
IF %QX1.4.0 AND NOT %QX1.5.19 AND ((%IX1.1.20 AND %ML2.1) OR (%IX1.1.21 AND %IX1.2.8) OR (%MX340 AND %IX1.2.59 AND NOT %IX1.1.21)) AND %ML100.10 THEN
    %WW150 := 0;
END_IF;

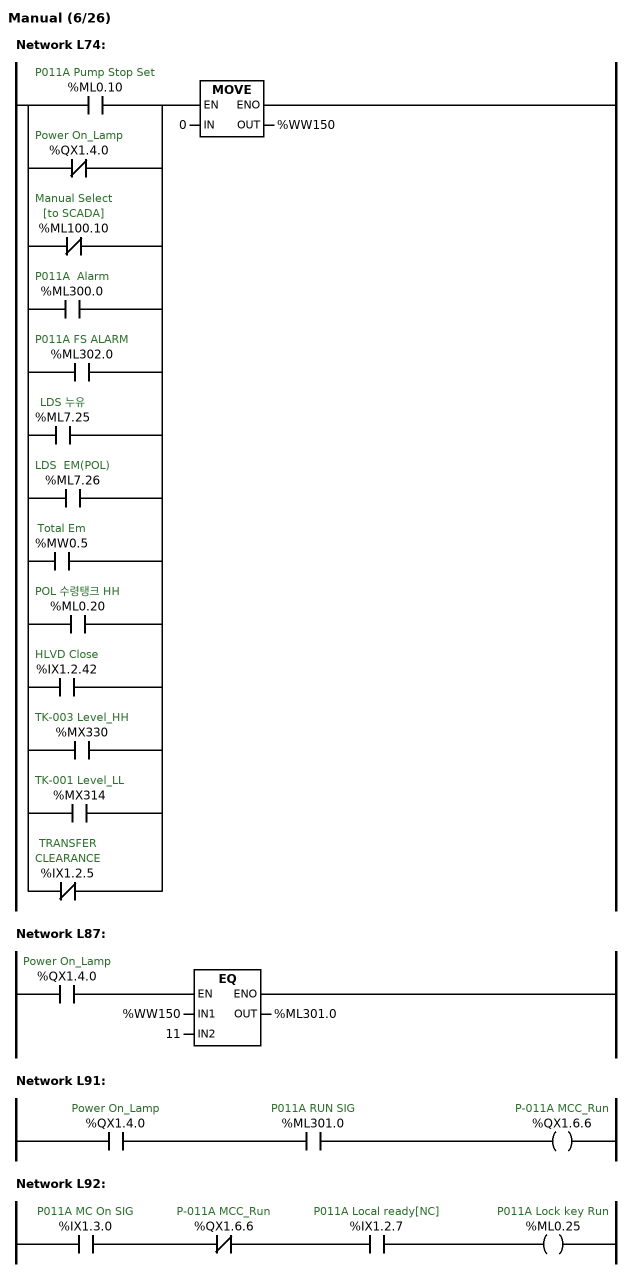
(* Rung L74 *)
IF %ML0.10 OR NOT %QX1.4.0 OR NOT %ML100.10 OR %ML300.0 OR %ML302.0 OR %ML7.25 OR %ML7.26 OR %MW0.5 OR %ML0.20 OR %IX1.2.42 OR %MX330 OR %MX314 OR NOT %IX1.2.5 THEN
    %WW150 := 0;
END_IF;
(* Rung L87 *)
IF %QX1.4.0 THEN %ML301.0 := %WW150 = 11; END_IF;
(* Rung L91 *)
%QX1.6.6 := %QX1.4.0 AND %ML301.0;
(* Rung L92 *)
%ML0.25 := %IX1.3.0 AND NOT %QX1.6.6 AND %IX1.2.7;

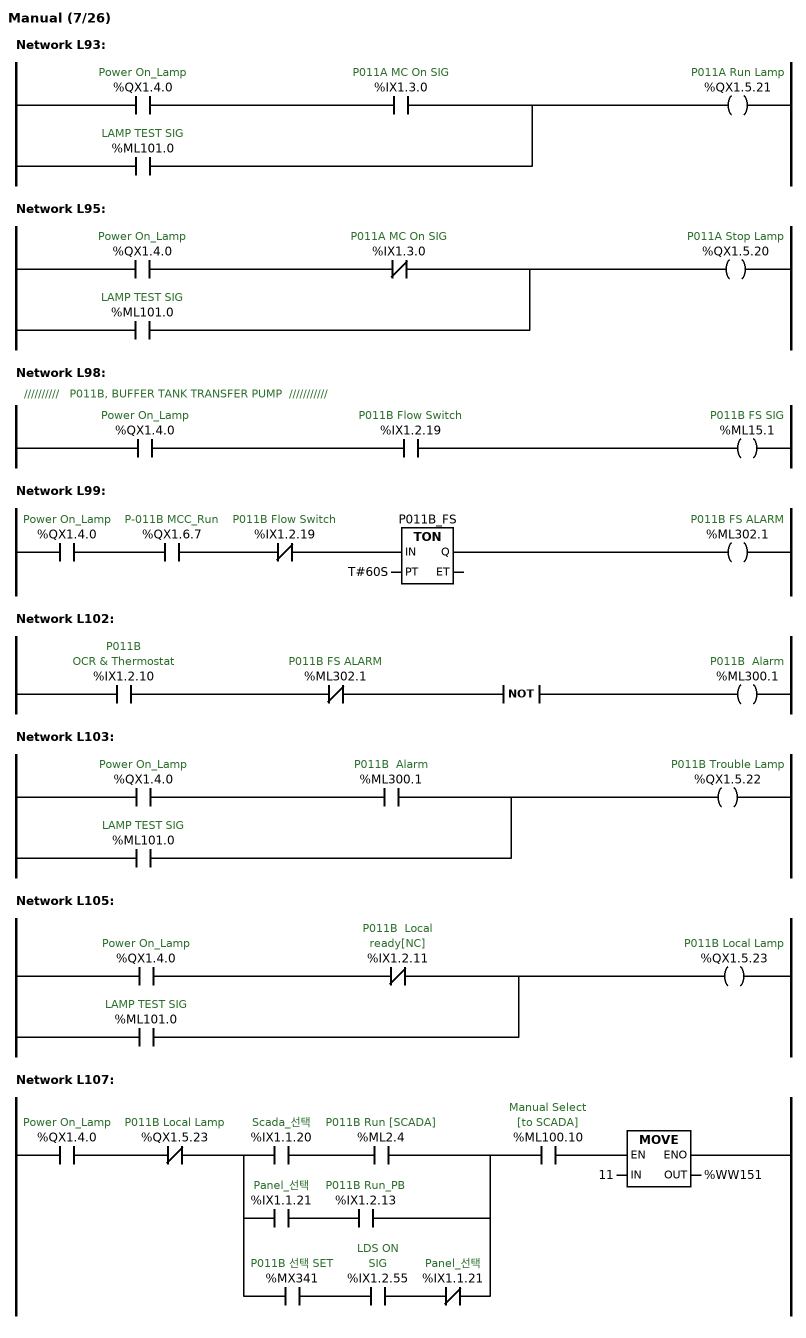
(* Rung L93 *)
%QX1.5.21 := (%QX1.4.0 AND %IX1.3.0) OR %ML101.0;
(* Rung L95 *)
%QX1.5.20 := (%QX1.4.0 AND NOT %IX1.3.0) OR %ML101.0;
(* //////////   P011B, BUFFER TANK TRANSFER PUMP  /////////// *)
(* Rung L98 *)
%ML15.1 := %QX1.4.0 AND %IX1.2.19;
(* Rung L99 *)
P011B_FS(IN := %QX1.4.0 AND %QX1.6.7 AND NOT %IX1.2.19, PT := T#60S);
%ML302.1 := P011B_FS.Q;
(* Rung L102 *)
%ML300.1 := NOT (%IX1.2.10 AND NOT %ML302.1);
(* Rung L103 *)
%QX1.5.22 := (%QX1.4.0 AND %ML300.1) OR %ML101.0;
(* Rung L105 *)
%QX1.5.23 := (%QX1.4.0 AND NOT %IX1.2.11) OR %ML101.0;
(* Rung L107 *)
IF %QX1.4.0 AND NOT %QX1.5.23 AND ((%IX1.1.20 AND %ML2.4) OR (%IX1.1.21 AND %IX1.2.13) OR (%MX341 AND %IX1.2.55 AND NOT %IX1.1.21)) AND %ML100.10 THEN
    %WW151 := 11;
END_IF;

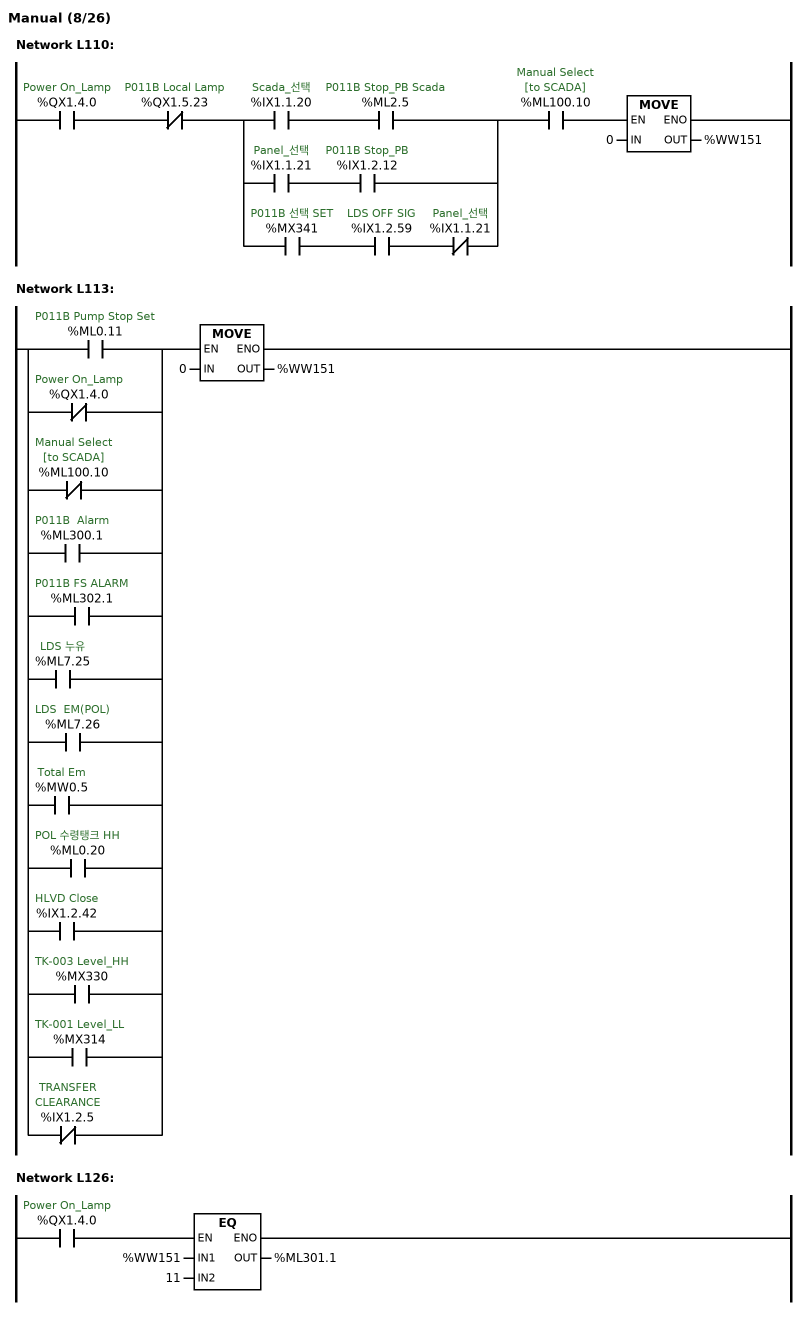
(* Rung L110 *)
IF %QX1.4.0 AND NOT %QX1.5.23 AND ((%IX1.1.20 AND %ML2.5) OR (%IX1.1.21 AND %IX1.2.12) OR (%MX341 AND %IX1.2.59 AND NOT %IX1.1.21)) AND %ML100.10 THEN
    %WW151 := 0;
END_IF;
(* Rung L113 *)
IF %ML0.11 OR NOT %QX1.4.0 OR NOT %ML100.10 OR %ML300.1 OR %ML302.1 OR %ML7.25 OR %ML7.26 OR %MW0.5 OR %ML0.20 OR %IX1.2.42 OR %MX330 OR %MX314 OR NOT %IX1.2.5 THEN
    %WW151 := 0;
END_IF;
(* Rung L126 *)
IF %QX1.4.0 THEN %ML301.1 := %WW151 = 11; END_IF;

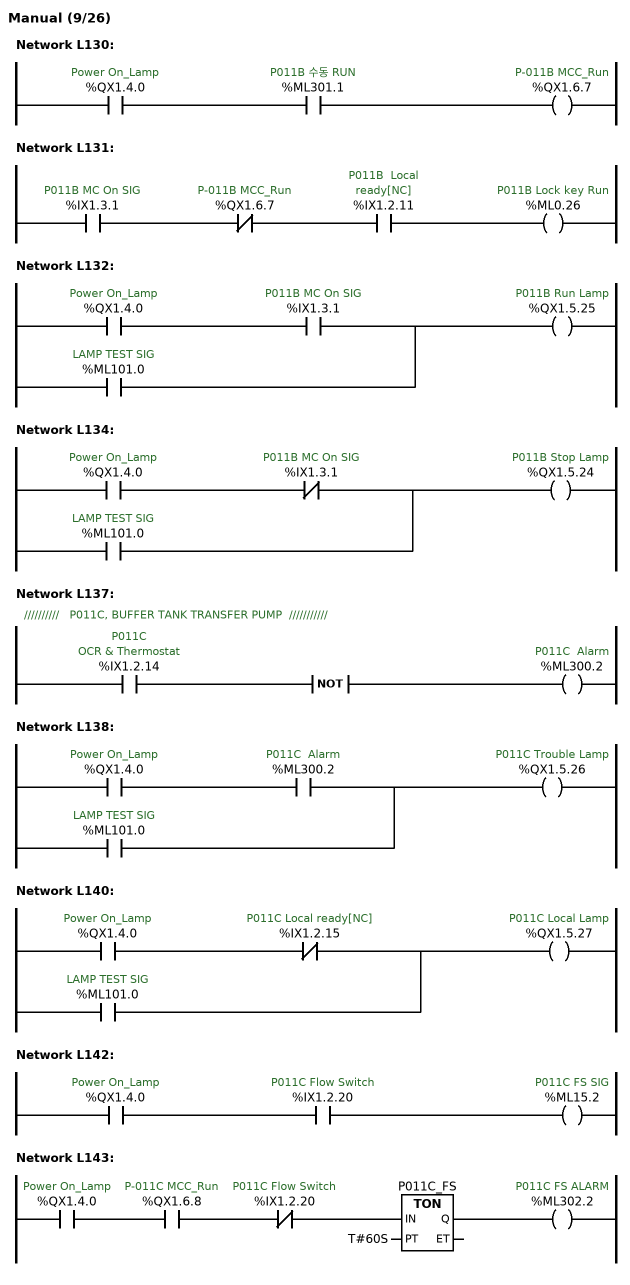
(* Rung L130 *)
%QX1.6.7 := %QX1.4.0 AND %ML301.1;
(* Rung L131 *)
%ML0.26 := %IX1.3.1 AND NOT %QX1.6.7 AND %IX1.2.11;
(* Rung L132 *)
%QX1.5.25 := (%QX1.4.0 AND %IX1.3.1) OR %ML101.0;
(* Rung L134 *)
%QX1.5.24 := (%QX1.4.0 AND NOT %IX1.3.1) OR %ML101.0;
(* //////////   P011C, BUFFER TANK TRANSFER PUMP  /////////// *)
(* Rung L137 *)
%ML300.2 := NOT %IX1.2.14;
(* Rung L138 *)
%QX1.5.26 := (%QX1.4.0 AND %ML300.2) OR %ML101.0;
(* Rung L140 *)
%QX1.5.27 := (%QX1.4.0 AND NOT %IX1.2.15) OR %ML101.0;
(* Rung L142 *)
%ML15.2 := %QX1.4.0 AND %IX1.2.20;
(* Rung L143 *)
P011C_FS(IN := %QX1.4.0 AND %QX1.6.8 AND NOT %IX1.2.20, PT := T#60S);
%ML302.2 := P011C_FS.Q;

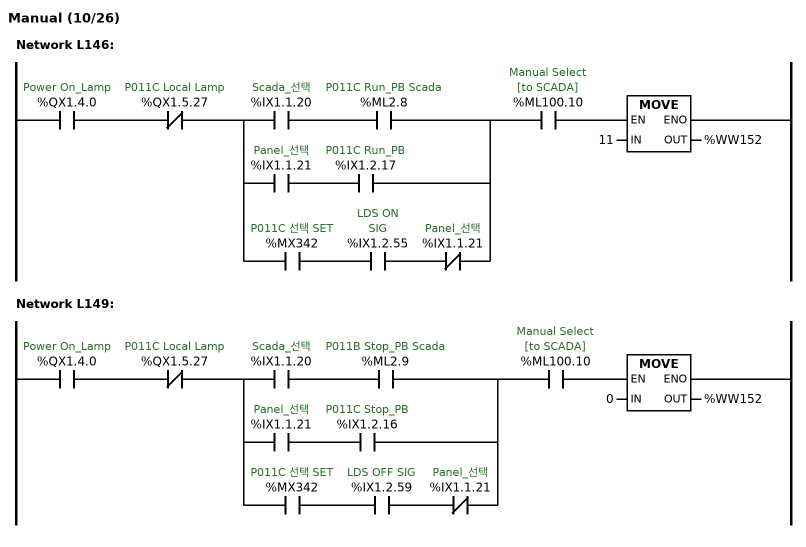
(* Rung L146 *)
IF %QX1.4.0 AND NOT %QX1.5.27 AND ((%IX1.1.20 AND %ML2.8) OR (%IX1.1.21 AND %IX1.2.17) OR (%MX342 AND %IX1.2.55 AND NOT %IX1.1.21)) AND %ML100.10 THEN
    %WW152 := 11;
END_IF;
(* Rung L149 *)
IF %QX1.4.0 AND NOT %QX1.5.27 AND ((%IX1.1.20 AND %ML2.9) OR (%IX1.1.21 AND %IX1.2.16) OR (%MX342 AND %IX1.2.59 AND NOT %IX1.1.21)) AND %ML100.10 THEN
    %WW152 := 0;
END_IF;

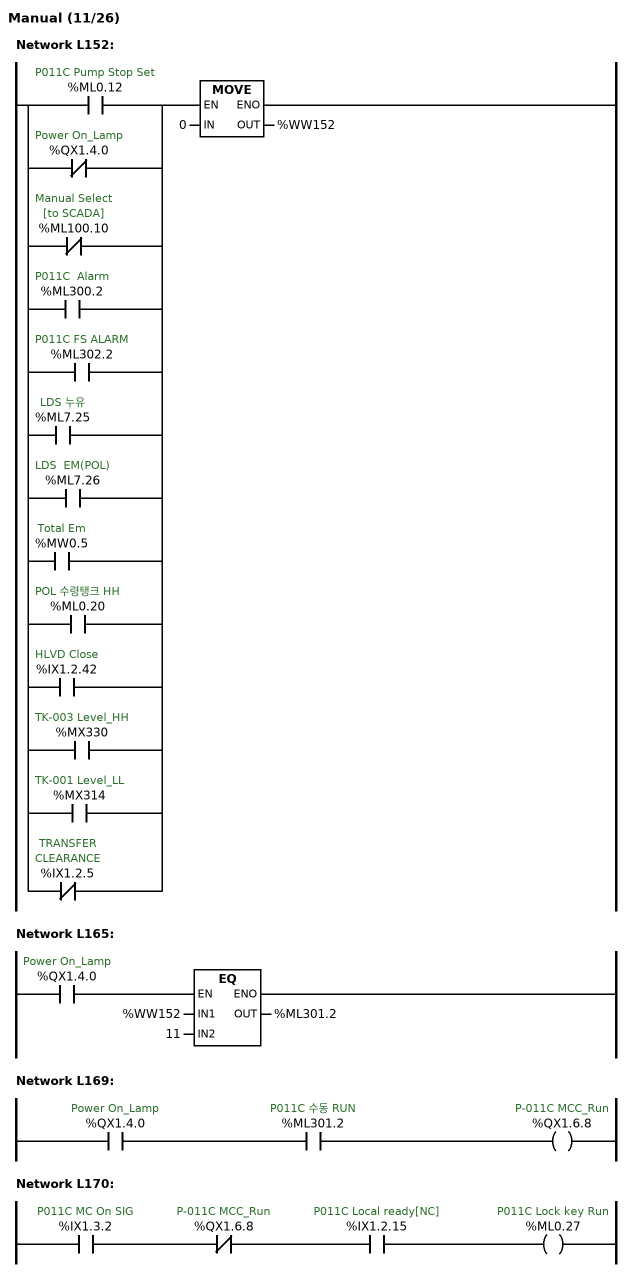
(* Rung L152 *)
IF %ML0.12 OR NOT %QX1.4.0 OR NOT %ML100.10 OR %ML300.2 OR %ML302.2 OR %ML7.25 OR %ML7.26 OR %MW0.5 OR %ML0.20 OR %IX1.2.42 OR %MX330 OR %MX314 OR NOT %IX1.2.5 THEN
    %WW152 := 0;
END_IF;
(* Rung L165 *)
IF %QX1.4.0 THEN %ML301.2 := %WW152 = 11; END_IF;
(* Rung L169 *)
%QX1.6.8 := %QX1.4.0 AND %ML301.2;
(* Rung L170 *)
%ML0.27 := %IX1.3.2 AND NOT %QX1.6.8 AND %IX1.2.15;

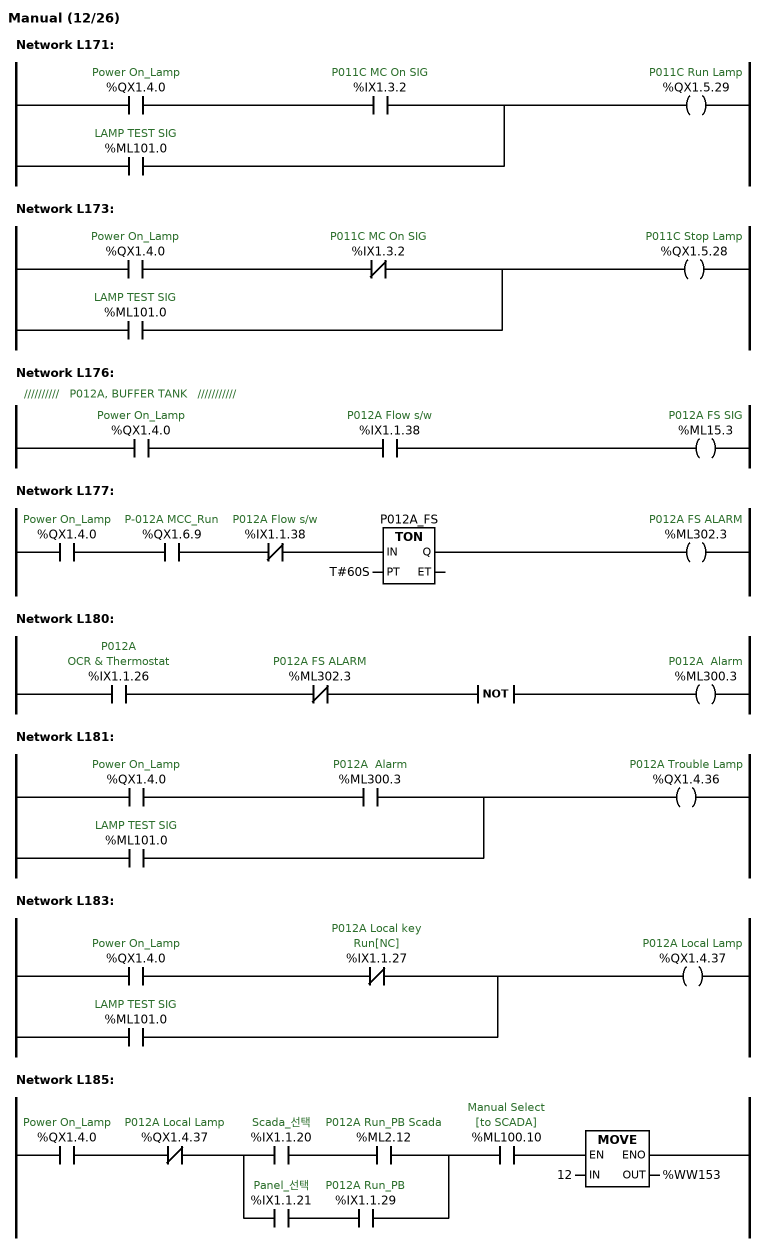
(* Rung L171 *)
%QX1.5.29 := (%QX1.4.0 AND %IX1.3.2) OR %ML101.0;
(* Rung L173 *)
%QX1.5.28 := (%QX1.4.0 AND NOT %IX1.3.2) OR %ML101.0;
(* //////////   P012A, BUFFER TANK   /////////// *)
(* Rung L176 *)
%ML15.3 := %QX1.4.0 AND %IX1.1.38;
(* Rung L177 *)
P012A_FS(IN := %QX1.4.0 AND %QX1.6.9 AND NOT %IX1.1.38, PT := T#60S);
%ML302.3 := P012A_FS.Q;
(* Rung L180 *)
%ML300.3 := NOT (%IX1.1.26 AND NOT %ML302.3);
(* Rung L181 *)
%QX1.4.36 := (%QX1.4.0 AND %ML300.3) OR %ML101.0;
(* Rung L183 *)
%QX1.4.37 := (%QX1.4.0 AND NOT %IX1.1.27) OR %ML101.0;
(* Rung L185 *)
IF %QX1.4.0 AND NOT %QX1.4.37 AND ((%IX1.1.20 AND %ML2.12) OR (%IX1.1.21 AND %IX1.1.29)) AND %ML100.10 THEN
    %WW153 := 12;
END_IF;

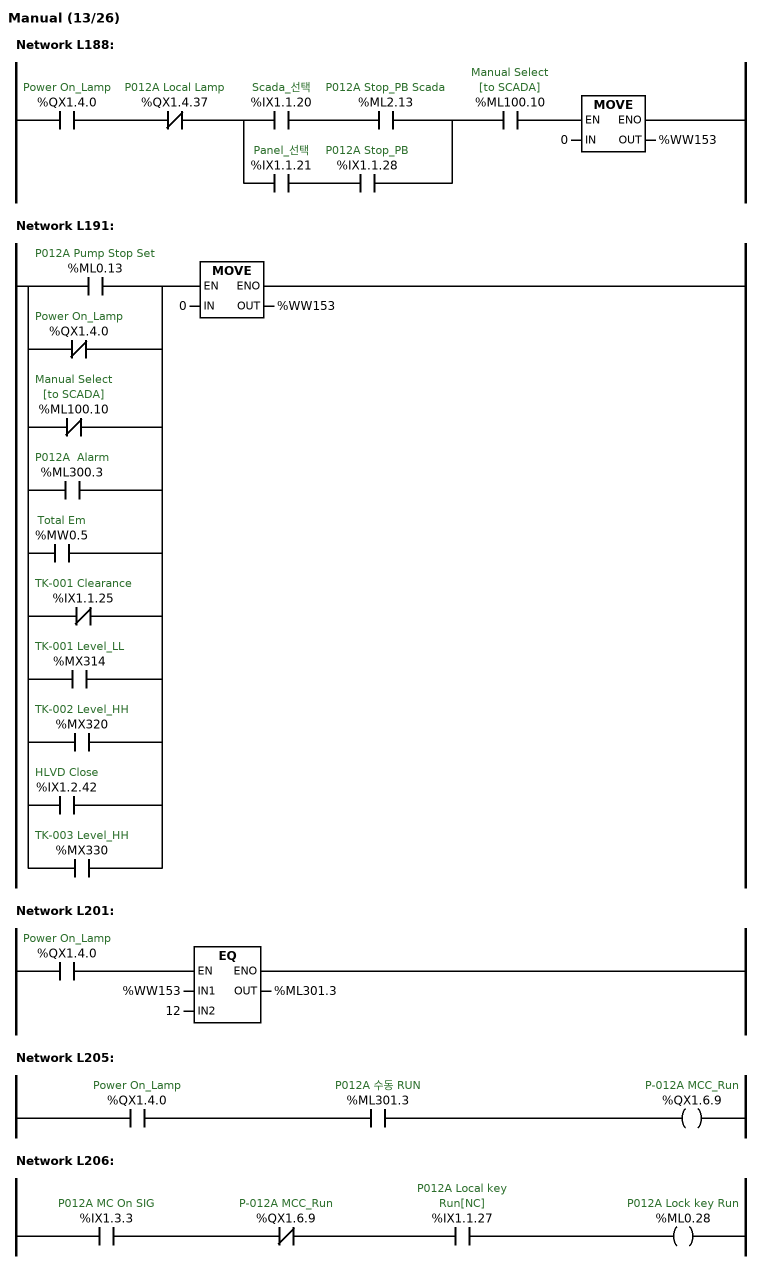
(* Rung L188 *)
IF %QX1.4.0 AND NOT %QX1.4.37 AND ((%IX1.1.20 AND %ML2.13) OR (%IX1.1.21 AND %IX1.1.28)) AND %ML100.10 THEN
    %WW153 := 0;
END_IF;
(* Rung L191 *)
IF %ML0.13 OR NOT %QX1.4.0 OR NOT %ML100.10 OR %ML300.3 OR %MW0.5 OR NOT %IX1.1.25 OR %MX314 OR %MX320 OR %IX1.2.42 OR %MX330 THEN
    %WW153 := 0;
END_IF;
(* Rung L201 *)
IF %QX1.4.0 THEN %ML301.3 := %WW153 = 12; END_IF;
(* Rung L205 *)
%QX1.6.9 := %QX1.4.0 AND %ML301.3;
(* Rung L206 *)
%ML0.28 := %IX1.3.3 AND NOT %QX1.6.9 AND %IX1.1.27;

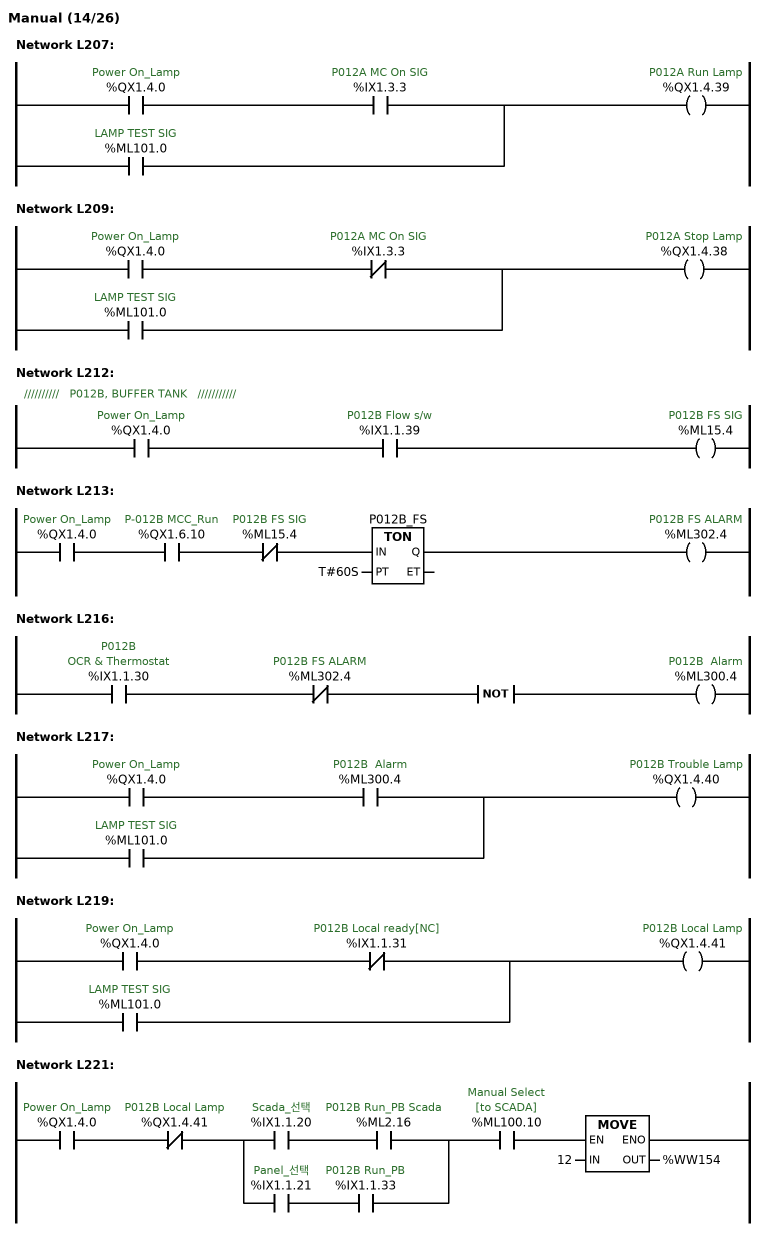
(* Rung L207 *)
%QX1.4.39 := (%QX1.4.0 AND %IX1.3.3) OR %ML101.0;
(* Rung L209 *)
%QX1.4.38 := (%QX1.4.0 AND NOT %IX1.3.3) OR %ML101.0;
(* //////////   P012B, BUFFER TANK   /////////// *)
(* Rung L212 *)
%ML15.4 := %QX1.4.0 AND %IX1.1.39;
(* Rung L213 *)
P012B_FS(IN := %QX1.4.0 AND %QX1.6.10 AND NOT %ML15.4, PT := T#60S);
%ML302.4 := P012B_FS.Q;
(* Rung L216 *)
%ML300.4 := NOT (%IX1.1.30 AND NOT %ML302.4);
(* Rung L217 *)
%QX1.4.40 := (%QX1.4.0 AND %ML300.4) OR %ML101.0;
(* Rung L219 *)
%QX1.4.41 := (%QX1.4.0 AND NOT %IX1.1.31) OR %ML101.0;
(* Rung L221 *)
IF %QX1.4.0 AND NOT %QX1.4.41 AND ((%IX1.1.20 AND %ML2.16) OR (%IX1.1.21 AND %IX1.1.33)) AND %ML100.10 THEN
    %WW154 := 12;
END_IF;

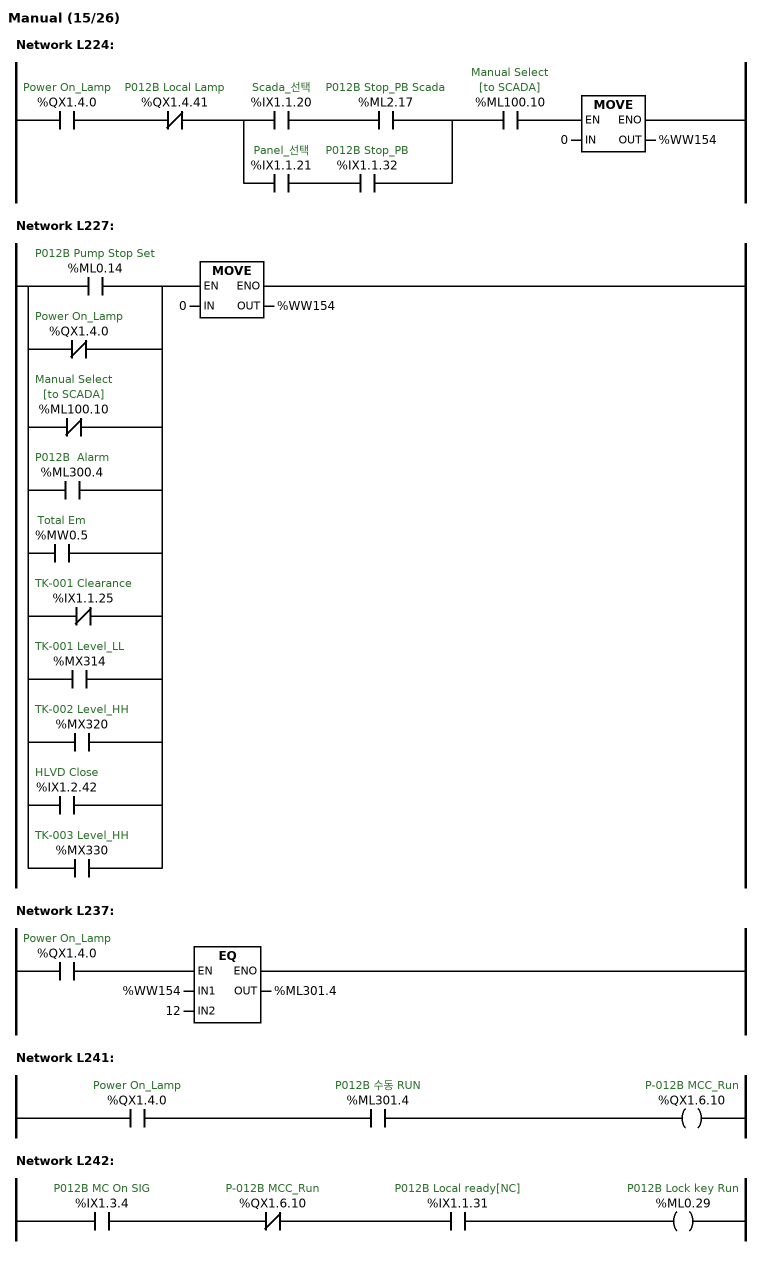
(* Rung L224 *)
IF %QX1.4.0 AND NOT %QX1.4.41 AND ((%IX1.1.20 AND %ML2.17) OR (%IX1.1.21 AND %IX1.1.32)) AND %ML100.10 THEN
    %WW154 := 0;
END_IF;
(* Rung L227 *)
IF %ML0.14 OR NOT %QX1.4.0 OR NOT %ML100.10 OR %ML300.4 OR %MW0.5 OR NOT %IX1.1.25 OR %MX314 OR %MX320 OR %IX1.2.42 OR %MX330 THEN
    %WW154 := 0;
END_IF;
(* Rung L237 *)
IF %QX1.4.0 THEN %ML301.4 := %WW154 = 12; END_IF;
(* Rung L241 *)
%QX1.6.10 := %QX1.4.0 AND %ML301.4;
(* Rung L242 *)
%ML0.29 := %IX1.3.4 AND NOT %QX1.6.10 AND %IX1.1.31;

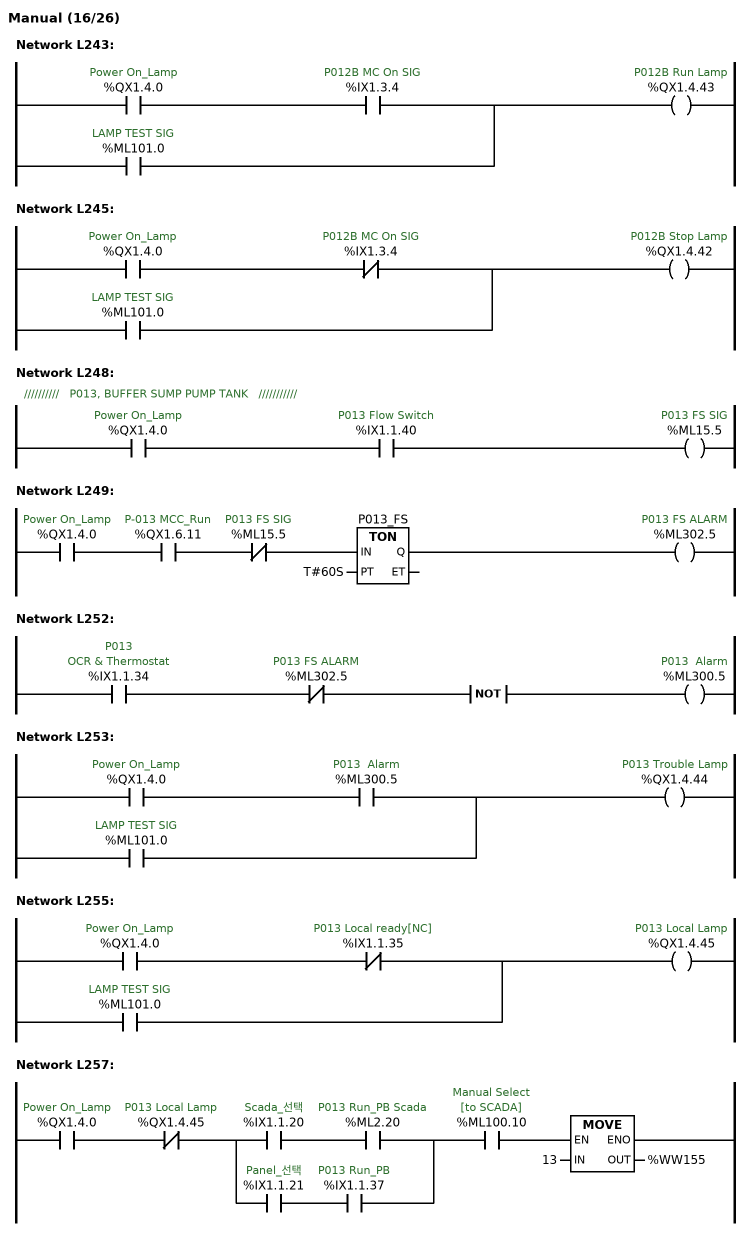
(* Rung L243 *)
%QX1.4.43 := (%QX1.4.0 AND %IX1.3.4) OR %ML101.0;
(* Rung L245 *)
%QX1.4.42 := (%QX1.4.0 AND NOT %IX1.3.4) OR %ML101.0;
(* //////////   P013, BUFFER SUMP PUMP TANK   /////////// *)
(* Rung L248 *)
%ML15.5 := %QX1.4.0 AND %IX1.1.40;
(* Rung L249 *)
P013_FS(IN := %QX1.4.0 AND %QX1.6.11 AND NOT %ML15.5, PT := T#60S);
%ML302.5 := P013_FS.Q;
(* Rung L252 *)
%ML300.5 := NOT (%IX1.1.34 AND NOT %ML302.5);
(* Rung L253 *)
%QX1.4.44 := (%QX1.4.0 AND %ML300.5) OR %ML101.0;
(* Rung L255 *)
%QX1.4.45 := (%QX1.4.0 AND NOT %IX1.1.35) OR %ML101.0;
(* Rung L257 *)
IF %QX1.4.0 AND NOT %QX1.4.45 AND ((%IX1.1.20 AND %ML2.20) OR (%IX1.1.21 AND %IX1.1.37)) AND %ML100.10 THEN
    %WW155 := 13;
END_IF;

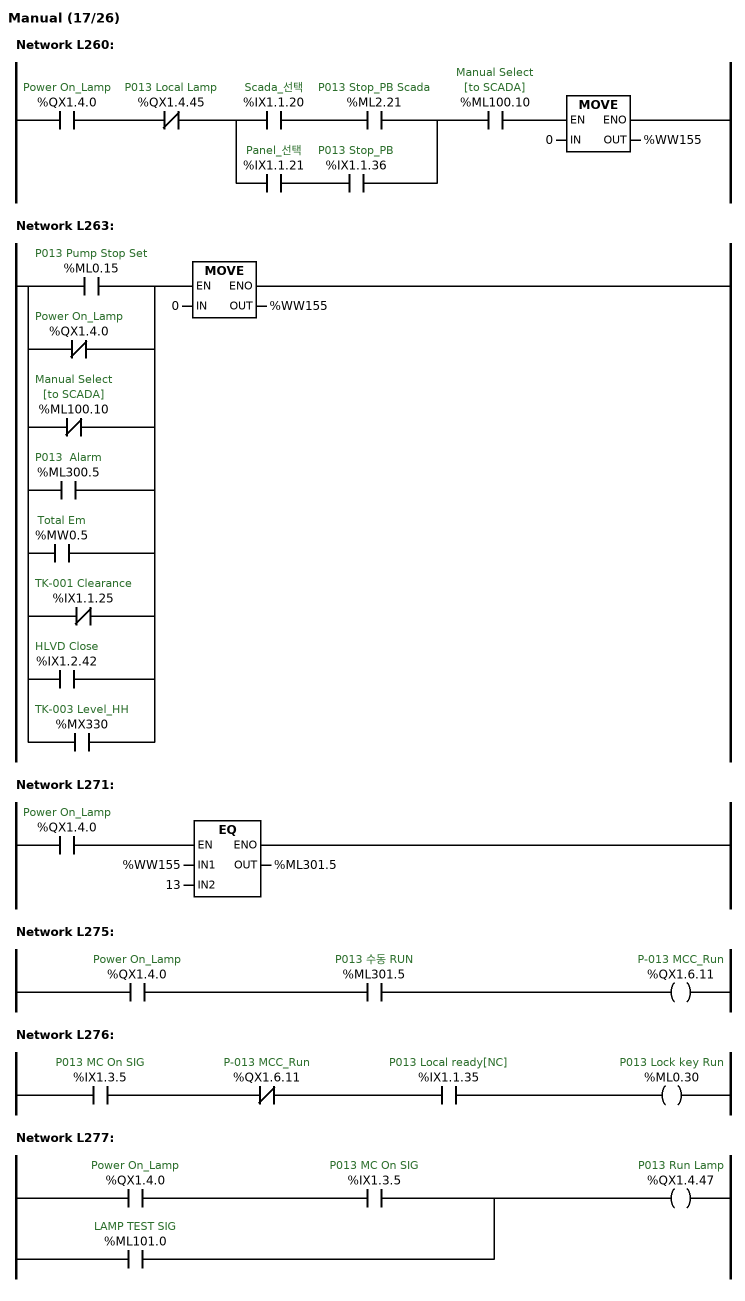
(* Rung L260 *)
IF %QX1.4.0 AND NOT %QX1.4.45 AND ((%IX1.1.20 AND %ML2.21) OR (%IX1.1.21 AND %IX1.1.36)) AND %ML100.10 THEN
    %WW155 := 0;
END_IF;
(* Rung L263 *)
IF %ML0.15 OR NOT %QX1.4.0 OR NOT %ML100.10 OR %ML300.5 OR %MW0.5 OR NOT %IX1.1.25 OR %IX1.2.42 OR %MX330 THEN
    %WW155 := 0;
END_IF;
(* Rung L271 *)
IF %QX1.4.0 THEN %ML301.5 := %WW155 = 13; END_IF;
(* Rung L275 *)
%QX1.6.11 := %QX1.4.0 AND %ML301.5;
(* Rung L276 *)
%ML0.30 := %IX1.3.5 AND NOT %QX1.6.11 AND %IX1.1.35;
(* Rung L277 *)
%QX1.4.47 := (%QX1.4.0 AND %IX1.3.5) OR %ML101.0;

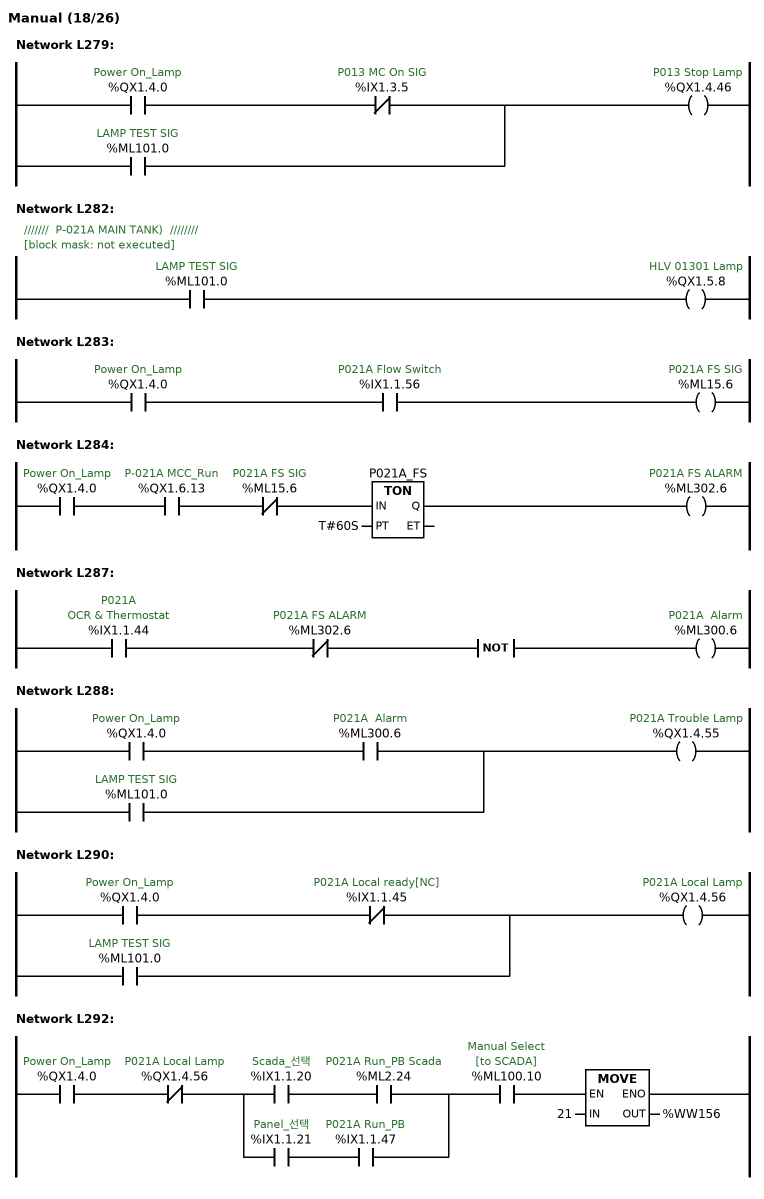
(* Rung L279 *)
%QX1.4.46 := (%QX1.4.0 AND NOT %IX1.3.5) OR %ML101.0;
(* ///////  P-021A MAIN TANK)  //////// *)
(* Rung L282 is block-masked: not executed *)
// %QX1.5.8 := %ML101.0;
(* Rung L283 *)
%ML15.6 := %QX1.4.0 AND %IX1.1.56;
(* Rung L284 *)
P021A_FS(IN := %QX1.4.0 AND %QX1.6.13 AND NOT %ML15.6, PT := T#60S);
%ML302.6 := P021A_FS.Q;
(* Rung L287 *)
%ML300.6 := NOT (%IX1.1.44 AND NOT %ML302.6);
(* Rung L288 *)
%QX1.4.55 := (%QX1.4.0 AND %ML300.6) OR %ML101.0;
(* Rung L290 *)
%QX1.4.56 := (%QX1.4.0 AND NOT %IX1.1.45) OR %ML101.0;
(* Rung L292 *)
IF %QX1.4.0 AND NOT %QX1.4.56 AND ((%IX1.1.20 AND %ML2.24) OR (%IX1.1.21 AND %IX1.1.47)) AND %ML100.10 THEN
    %WW156 := 21;
END_IF;

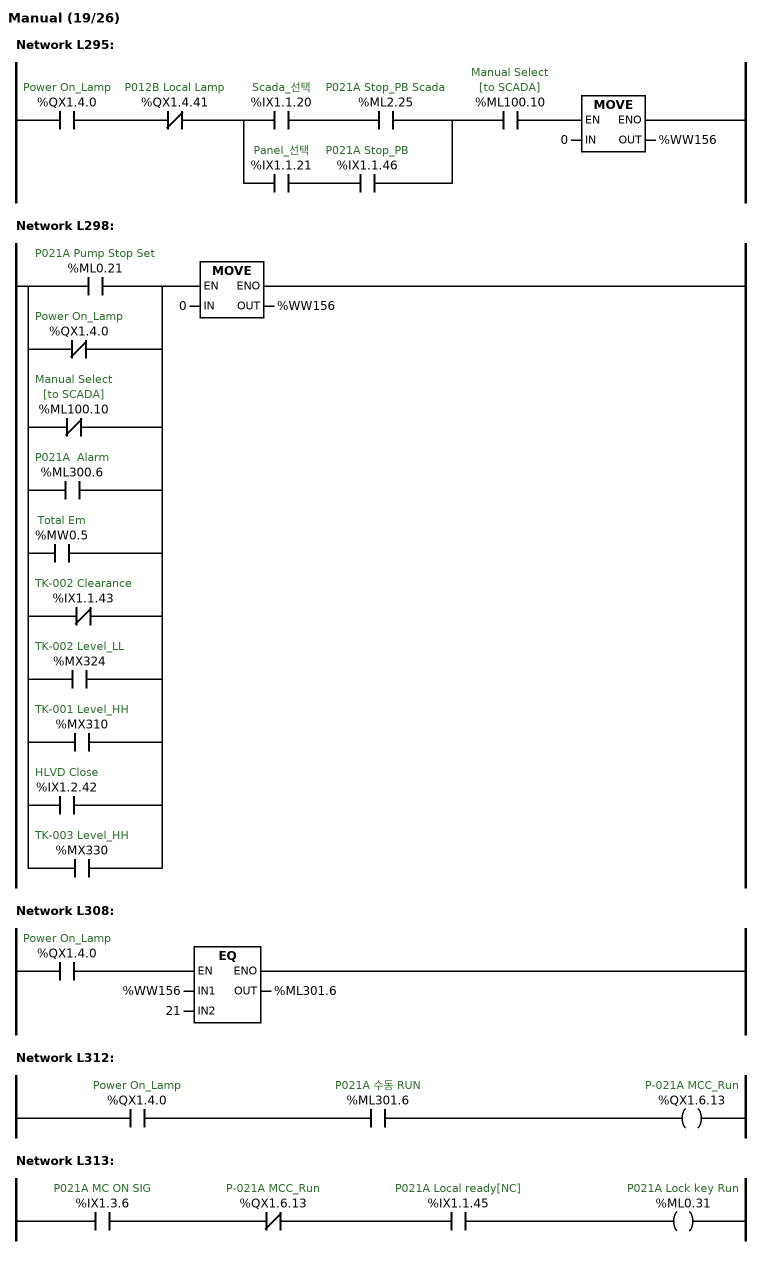
(* Rung L295 *)
IF %QX1.4.0 AND NOT %QX1.4.41 AND ((%IX1.1.20 AND %ML2.25) OR (%IX1.1.21 AND %IX1.1.46)) AND %ML100.10 THEN
    %WW156 := 0;
END_IF;
(* Rung L298 *)
IF %ML0.21 OR NOT %QX1.4.0 OR NOT %ML100.10 OR %ML300.6 OR %MW0.5 OR NOT %IX1.1.43 OR %MX324 OR %MX310 OR %IX1.2.42 OR %MX330 THEN
    %WW156 := 0;
END_IF;
(* Rung L308 *)
IF %QX1.4.0 THEN %ML301.6 := %WW156 = 21; END_IF;
(* Rung L312 *)
%QX1.6.13 := %QX1.4.0 AND %ML301.6;
(* Rung L313 *)
%ML0.31 := %IX1.3.6 AND NOT %QX1.6.13 AND %IX1.1.45;

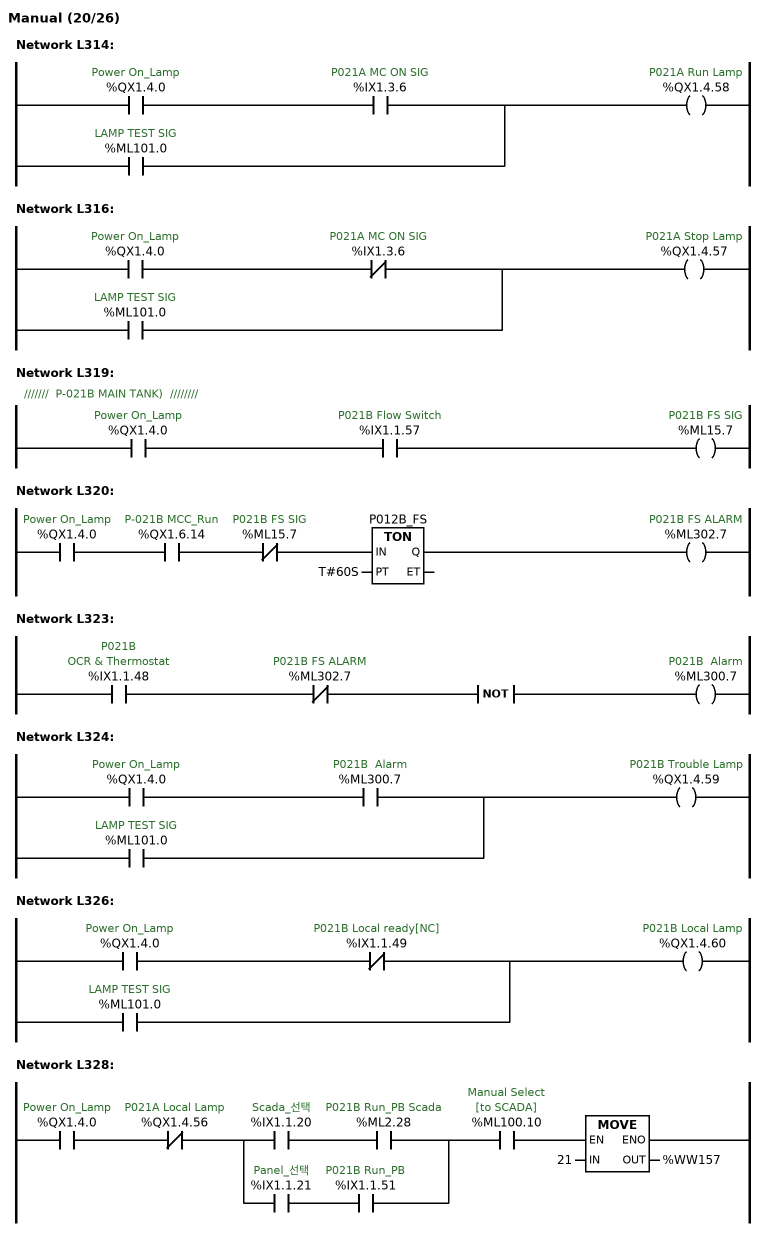
(* Rung L314 *)
%QX1.4.58 := (%QX1.4.0 AND %IX1.3.6) OR %ML101.0;
(* Rung L316 *)
%QX1.4.57 := (%QX1.4.0 AND NOT %IX1.3.6) OR %ML101.0;
(* ///////  P-021B MAIN TANK)  //////// *)
(* Rung L319 *)
%ML15.7 := %QX1.4.0 AND %IX1.1.57;
(* Rung L320 *)
P012B_FS(IN := %QX1.4.0 AND %QX1.6.14 AND NOT %ML15.7, PT := T#60S);
%ML302.7 := P012B_FS.Q;
(* Rung L323 *)
%ML300.7 := NOT (%IX1.1.48 AND NOT %ML302.7);
(* Rung L324 *)
%QX1.4.59 := (%QX1.4.0 AND %ML300.7) OR %ML101.0;
(* Rung L326 *)
%QX1.4.60 := (%QX1.4.0 AND NOT %IX1.1.49) OR %ML101.0;
(* Rung L328 *)
IF %QX1.4.0 AND NOT %QX1.4.56 AND ((%IX1.1.20 AND %ML2.28) OR (%IX1.1.21 AND %IX1.1.51)) AND %ML100.10 THEN
    %WW157 := 21;
END_IF;

